LIN {X 0,Y 298.465,Z 418.303,A -85,B 0,C 180,E1 -16416.814,E2 -16416.814} C_VEL
LIN {X 0,Y 298.452,Z 418.307,A -85,B 0,C 180,E1 -16421.25,E2 -16421.25} C_VEL
LIN {X 0,Y 298.485,Z 418.303,A -85,B 0,C 180,E1 -16425.061,E2 -16425.061} C_VEL
LIN {X 0,Y 298.449,Z 418.307,A -85,B 0,C 180,E1 -16428.898,E2 -16428.898} C_VEL
LIN {X 0,Y 298.467,Z 418.307,A -85,B 0,C 180,E1 -16433.187,E2 -16433.187} C_VEL
LIN {X 0,Y 298.392,Z 418.317,A -85,B 0,C 180,E1 -16437.201,E2 -16437.201} C_VEL
LIN {X 0,Y 298.467,Z 418.305,A -85,B 0,C 180,E1 -16441.906,E2 -16441.906} C_VEL
LIN {X 0,Y 298.473,Z 418.306,A -85,B 0,C 180,E1 -16444.924,E2 -16444.924} C_VEL
LIN {X 0,Y 298.363,Z 418.483,A -85,B 0,C 180,E1 -16449.129,E2 -16449.129} C_VEL
LIN {X 0,Y 297.959,Z 422.878,A -85,B 0,C 180,E1 -16453.559,E2 -16453.559} C_VEL
LIN {X 0,Y 297.845,Z 425.727,A -85,B 0,C 180,E1 -16456.352,E2 -16456.352} C_VEL
LIN {X 0,Y 297.552,Z 430.816,A -85,B 0,C 180,E1 -16461.168,E2 -16461.168} C_VEL
LIN {X 0,Y 297.561,Z 431.032,A -85,B 0,C 180,E1 -16461.37,E2 -16461.37} C_VEL
LIN {X 0,Y 300.495,Z 443.519,A -85,B 0,C 180,E1 -16462.124,E2 -16462.124} C_VEL
LIN {X 0,Y 302.874,Z 456.628,A -85,B 0,C 180,E1 -16463.149,E2 -16463.149} C_VEL
LIN {X 0,Y 304.31,Z 467.202,A -85,B 0,C 180,E1 -16464.177,E2 -16464.177} C_VEL
LIN {X 0,Y 303.211,Z 477.949,A -85,B 0,C 180,E1 -16465.327,E2 -16465.327} C_VEL
LIN {X 0,Y 301.899,Z 489.013,A -85,B 0,C 180,E1 -16466.831,E2 -16466.831} C_VEL
LIN {X 0,Y 300.698,Z 497.91,A -85,B 0,C 180,E1 -16468.326,E2 -16468.326} C_VEL
LIN {X 0,Y 299.564,Z 506.081,A -85,B 0,C 180,E1 -16470,E2 -16470} C_VEL
LIN {X 0,Y 298.454,Z 514.101,A -85,B 0,C 180,E1 -16472.024,E2 -16472.024} C_VEL
LIN {X 0,Y 297.678,Z 520.511,A -85,B 0,C 180,E1 -16474.062,E2 -16474.062} C_VEL
LIN {X 0,Y 297.162,Z 525.845,A -85,B 0,C 180,E1 -16476.228,E2 -16476.228} C_VEL
LIN {X 0,Y 296.792,Z 529.552,A -85,B 0,C 180,E1 -16478.168,E2 -16478.168} C_VEL
LIN {X 0,Y 296.549,Z 531.596,A -85,B 0,C 180,E1 -16479.549,E2 -16479.549} C_VEL
LIN {X 0,Y 296.405,Z 533.217,A -85,B 0,C 180,E1 -16480.935,E2 -16480.935} C_VEL
LIN {X 0,Y 296.357,Z 535.085,A -85,B 0,C 180,E1 -16483.518,E2 -16483.518} C_VEL
LIN {X 0,Y 296.332,Z 535.507,A -85,B 0,C 180,E1 -16485.122,E2 -16485.122} C_VEL
LIN {X 0,Y 296.381,Z 535.459,A -85,B 0,C 180,E1 -16486.532,E2 -16486.532} C_VEL
LIN {X 0,Y 296.708,Z 534.552,A -85,B 0,C 180,E1 -16488.655,E2 -16488.655} C_VEL
LIN {X 0,Y 297.131,Z 532.679,A -85,B 0,C 180,E1 -16490.781,E2 -16490.781} C_VEL
LIN {X 0,Y 297.877,Z 529.561,A -85,B 0,C 180,E1 -16493.052,E2 -16493.052} C_VEL
LIN {X 0,Y 298.727,Z 525.744,A -85,B 0,C 180,E1 -16495.054,E2 -16495.054} C_VEL
LIN {X 0,Y 300.094,Z 519.861,A -85,B 0,C 180,E1 -16497.39,E2 -16497.39} C_VEL
LIN {X 0,Y 301.823,Z 512.406,A -85,B 0,C 180,E1 -16499.657,E2 -16499.657} C_VEL
LIN {X 0,Y 303.322,Z 505.485,A -85,B 0,C 180,E1 -16501.343,E2 -16501.343} C_VEL
LIN {X 0,Y 305.278,Z 496.379,A -85,B 0,C 180,E1 -16503.145,E2 -16503.145} C_VEL
LIN {X 0,Y 307.219,Z 486.66,A -85,B 0,C 180,E1 -16504.674,E2 -16504.674} C_VEL
LIN {X 0,Y 309.046,Z 475.83,A -85,B 0,C 180,E1 -16506.045,E2 -16506.045} C_VEL
LIN {X 0,Y 309.437,Z 473.03,A -85,B 0,C 180,E1 -16506.356,E2 -16506.356} C_VEL
LIN {X 0,Y 307.623,Z 462.047,A -85,B 0,C 180,E1 -16507.717,E2 -16507.717} C_VEL
LIN {X 0,Y 304.42,Z 449.779,A -85,B 0,C 180,E1 -16509.079,E2 -16509.079} C_VEL
LIN {X 0,Y 300.228,Z 437.616,A -85,B 0,C 180,E1 -16510.282,E2 -16510.282} C_VEL
LIN {X 0,Y 298.18,Z 432.147,A -85,B 0,C 180,E1 -16510.762,E2 -16510.762} C_VEL
LIN {X 0,Y 298.092,Z 431.637,A -85,B 0,C 180,E1 -16510.836,E2 -16510.836} C_VEL
LIN {X 0,Y 298.317,Z 429.506,A -85,B 0,C 180,E1 -16513.094,E2 -16513.094} C_VEL
LIN {X 0,Y 298.674,Z 426.006,A -85,B 0,C 180,E1 -16516.97,E2 -16516.97} C_VEL
LIN {X 0,Y 298.862,Z 424.41,A -85,B 0,C 180,E1 -16518.819,E2 -16518.819} C_VEL
LIN {X 0,Y 298.783,Z 421.553,A -85,B 0,C 180,E1 -16522.297,E2 -16522.297} C_VEL
LIN {X 0,Y 298.537,Z 419.047,A -85,B 0,C 180,E1 -16525.598,E2 -16525.598} C_VEL
LIN {X 0,Y 298.394,Z 418.32,A -85,B 0,C 180,E1 -16527.2,E2 -16527.2} C_VEL
LIN {X 0,Y 298.429,Z 418.312,A -85,B 0,C 180,E1 -16530.614,E2 -16530.614} C_VEL
LIN {X 0,Y 298.48,Z 418.307,A -85,B 0,C 180,E1 -16533.474,E2 -16533.474} C_VEL
LIN {X 0,Y 298.427,Z 418.313,A -85,B 0,C 180,E1 -16536.699,E2 -16536.699} C_VEL
LIN {X 0,Y 298.534,Z 418.296,A -85,B 0,C 180,E1 -16540.757,E2 -16540.757} C_VEL
LIN {X 0,Y 298.589,Z 418.291,A -85,B 0,C 180,E1 -16544.995,E2 -16544.995} C_VEL
LIN {X 0,Y 298.589,Z 418.287,A -85,B 0,C 180,E1 -16549.147,E2 -16549.147} C_VEL
LIN {X 0,Y 298.749,Z 418.27,A -85,B 0,C 180,E1 -16552.391,E2 -16552.391} C_VEL
LIN {X 0,Y 298.091,Z 418.355,A -85,B 0,C 180,E1 -16553.514,E2 -16553.514} C_VEL
LIN {X 0,Y 295.235,Z 418.71,A -85,B 0,C 180,E1 -16555.344,E2 -16555.344} C_VEL
LIN {X 0,Y 292.852,Z 419.006,A -85,B 0,C 180,E1 -16556.829,E2 -16556.829} C_VEL
LIN {X 0,Y 291.896,Z 419.127,A -85,B 0,C 180,E1 -16557.979,E2 -16557.979} C_VEL
LIN {X 0,Y 291.854,Z 419.128,A -85,B 0,C 180,E1 -16558.368,E2 -16558.368} C_VEL
LIN {X 0,Y 291.887,Z 419.128,A -85,B 0,C 180,E1 -16561.38,E2 -16561.38} C_VEL
LIN {X 0,Y 291.738,Z 419.14,A -85,B 0,C 180,E1 -16566.918,E2 -16566.918} C_VEL
LIN {X 0,Y 291.626,Z 419.161,A -85,B 0,C 180,E1 -16569.712,E2 -16569.712} C_VEL
LIN {X 0,Y 291.519,Z 419.172,A -85,B 0,C 180,E1 -16573.951,E2 -16573.951} C_VEL
LIN {X 0,Y 291.484,Z 419.179,A -85,B 0,C 180,E1 -16576.818,E2 -16576.818} C_VEL
LIN {X 0,Y 291.448,Z 419.185,A -85,B 0,C 180,E1 -16579.875,E2 -16579.875} C_VEL
LIN {X 0,Y 291.398,Z 419.19,A -85,B 0,C 180,E1 -16584.206,E2 -16584.206} C_VEL
LIN {X 0,Y 291.42,Z 419.187,A -85,B 0,C 180,E1 -16587.272,E2 -16587.272} C_VEL
LIN {X 0,Y 291.335,Z 419.197,A -85,B 0,C 180,E1 -16590.437,E2 -16590.437} C_VEL
LIN {X 0,Y 291.343,Z 419.194,A -85,B 0,C 180,E1 -16593.699,E2 -16593.699} C_VEL
LIN {X 0,Y 291.37,Z 419.185,A -85,B 0,C 180,E1 -16597.254,E2 -16597.254} C_VEL
LIN {X 0,Y 291.358,Z 419.241,A -85,B 0,C 180,E1 -16598.412,E2 -16598.412} C_VEL
LIN {X 0,Y 291.799,Z 422.011,A -85,B 0,C 180,E1 -16601.701,E2 -16601.701} C_VEL
LIN {X 0,Y 292.466,Z 425.825,A -85,B 0,C 180,E1 -16605.824,E2 -16605.824} C_VEL
LIN {X 0,Y 293.109,Z 429.691,A -85,B 0,C 180,E1 -16609.655,E2 -16609.655} C_VEL
LIN {X 0,Y 293.444,Z 433.625,A -85,B 0,C 180,E1 -16613.22,E2 -16613.22} C_VEL
LIN {X 0,Y 293.338,Z 435.615,A -85,B 0,C 180,E1 -16614.9,E2 -16614.9} C_VEL
LIN {X 0,Y 292.657,Z 439.593,A -85,B 0,C 180,E1 -16618.109,E2 -16618.109} C_VEL
LIN {X 0,Y 291.708,Z 445.236,A -85,B 0,C 180,E1 -16622.467,E2 -16622.467} C_VEL
LIN {X 0,Y 292.691,Z 448.629,A -85,B 0,C 180,E1 -16622.729,E2 -16622.729} C_VEL
LIN {X 0,Y 296.821,Z 462.357,A -85,B 0,C 180,E1 -16623.972,E2 -16623.972} C_VEL
LIN {X 0,Y 299.378,Z 474.172,A -85,B 0,C 180,E1 -16625.182,E2 -16625.182} C_VEL
LIN {X 0,Y 300.89,Z 486.394,A -85,B 0,C 180,E1 -16626.605,E2 -16626.605} C_VEL
LIN {X 0,Y 301.175,Z 494.957,A -85,B 0,C 180,E1 -16627.716,E2 -16627.716} C_VEL
LIN {X 0,Y 299.107,Z 505.649,A -85,B 0,C 180,E1 -16629.183,E2 -16629.183} C_VEL
LIN {X 0,Y 297.197,Z 514.413,A -85,B 0,C 180,E1 -16630.667,E2 -16630.667} C_VEL
LIN {X 0,Y 295.502,Z 522.486,A -85,B 0,C 180,E1 -16632.348,E2 -16632.348} C_VEL
LIN {X 0,Y 293.7,Z 530.437,A -85,B 0,C 180,E1 -16634.383,E2 -16634.383} C_VEL
LIN {X 0,Y 292.338,Z 535.848,A -85,B 0,C 180,E1 -16636.089,E2 -16636.089} C_VEL
LIN {X 0,Y 291.19,Z 541.166,A -85,B 0,C 180,E1 -16638.162,E2 -16638.162} C_VEL
LIN {X 0,Y 290.341,Z 545.336,A -85,B 0,C 180,E1 -16640.245,E2 -16640.245} C_VEL
LIN {X 0,Y 289.928,Z 547.557,A -85,B 0,C 180,E1 -16641.637,E2 -16641.637} C_VEL
LIN {X 0,Y 289.673,Z 549.306,A -85,B 0,C 180,E1 -16643.032,E2 -16643.032} C_VEL
LIN {X 0,Y 289.406,Z 551.603,A -85,B 0,C 180,E1 -16645.822,E2 -16645.822} C_VEL
LIN {X 0,Y 289.432,Z 552.172,A -85,B 0,C 180,E1 -16647.216,E2 -16647.216} C_VEL
LIN {X 0,Y 289.415,Z 552.31,A -85,B 0,C 180,E1 -16648.608,E2 -16648.608} C_VEL
LIN {X 0,Y 289.438,Z 552.054,A -85,B 0,C 180,E1 -16650,E2 -16650} C_VEL
LIN {X 0,Y 289.421,Z 551.408,A -85,B 0,C 180,E1 -16651.391,E2 -16651.391} C_VEL
LIN {X 0,Y 289.467,Z 550.372,A -85,B 0,C 180,E1 -16652.783,E2 -16652.783} C_VEL
LIN {X 0,Y 289.434,Z 548.879,A -85,B 0,C 180,E1 -16654.177,E2 -16654.177} C_VEL
LIN {X 0,Y 289.554,Z 545.838,A -85,B 0,C 180,E1 -16656.27,E2 -16656.27} C_VEL
LIN {X 0,Y 289.851,Z 541.724,A -85,B 0,C 180,E1 -16658.365,E2 -16658.365} C_VEL
LIN {X 0,Y 290.47,Z 535.4,A -85,B 0,C 180,E1 -16660.807,E2 -16660.807} C_VEL
LIN {X 0,Y 291.304,Z 528.501,A -85,B 0,C 180,E1 -16662.894,E2 -16662.894} C_VEL
LIN {X 0,Y 292.264,Z 521.451,A -85,B 0,C 180,E1 -16664.624,E2 -16664.624} C_VEL
LIN {X 0,Y 293.456,Z 512.95,A -85,B 0,C 180,E1 -16666.343,E2 -16666.343} C_VEL
LIN {X 0,Y 294.727,Z 502.406,A -85,B 0,C 180,E1 -16668.058,E2 -16668.058} C_VEL
LIN {X 0,Y 296.106,Z 491.99,A -85,B 0,C 180,E1 -16669.407,E2 -16669.407} C_VEL
LIN {X 0,Y 296.167,Z 487.329,A -85,B 0,C 180,E1 -16669.944,E2 -16669.944} C_VEL
LIN {X 0,Y 295.093,Z 475.372,A -85,B 0,C 180,E1 -16671.174,E2 -16671.174} C_VEL
LIN {X 0,Y 293.48,Z 462.982,A -85,B 0,C 180,E1 -16672.178,E2 -16672.178} C_VEL
LIN {X 0,Y 291.441,Z 450.758,A -85,B 0,C 180,E1 -16672.935,E2 -16672.935} C_VEL
LIN {X 0,Y 290.549,Z 445.893,A -85,B 0,C 180,E1 -16673.194,E2 -16673.194} C_VEL
LIN {X 0,Y 291.111,Z 440.04,A -85,B 0,C 180,E1 -16677.302,E2 -16677.302} C_VEL
LIN {X 0,Y 292.02,Z 433.549,A -85,B 0,C 180,E1 -16681.969,E2 -16681.969} C_VEL
LIN {X 0,Y 292.587,Z 429.133,A -85,B 0,C 180,E1 -16685.245,E2 -16685.245} C_VEL
LIN {X 0,Y 292.659,Z 426.105,A -85,B 0,C 180,E1 -16687.583,E2 -16687.583} C_VEL
LIN {X 0,Y 291.783,Z 421.133,A -85,B 0,C 180,E1 -16691.696,E2 -16691.696} C_VEL
LIN {X 0,Y 291.441,Z 419.183,A -85,B 0,C 180,E1 -16693.518,E2 -16693.518} C_VEL
LIN {X 0,Y 291.337,Z 419.196,A -85,B 0,C 180,E1 -16697.51,E2 -16697.51} C_VEL
LIN {X 0,Y 291.349,Z 419.196,A -85,B 0,C 180,E1 -16701.157,E2 -16701.157} C_VEL
LIN {X 0,Y 291.357,Z 419.193,A -85,B 0,C 180,E1 -16704.625,E2 -16704.625} C_VEL
LIN {X 0,Y 291.367,Z 419.188,A -85,B 0,C 180,E1 -16707.95,E2 -16707.95} C_VEL
LIN {X 0,Y 291.377,Z 419.184,A -85,B 0,C 180,E1 -16711.158,E2 -16711.158} C_VEL
LIN {X 0,Y 291.411,Z 419.181,A -85,B 0,C 180,E1 -16714.271,E2 -16714.271} C_VEL
LIN {X 0,Y 291.376,Z 419.188,A -85,B 0,C 180,E1 -16717.299,E2 -16717.299} C_VEL
LIN {X 0,Y 291.452,Z 419.178,A -85,B 0,C 180,E1 -16720.269,E2 -16720.269} C_VEL
LIN {X 0,Y 291.51,Z 419.167,A -85,B 0,C 180,E1 -16724.652,E2 -16724.652} C_VEL
LIN {X 0,Y 291.53,Z 419.17,A -85,B 0,C 180,E1 -16728.88,E2 -16728.88} C_VEL
LIN {X 0,Y 291.704,Z 419.146,A -85,B 0,C 180,E1 -16731.688,E2 -16731.688} C_VEL
LIN {X 0,Y 291.627,Z 419.154,A -85,B 0,C 180,E1 -16734.468,E2 -16734.468} C_VEL
LIN {X 0,Y 291.884,Z 419.122,A -85,B 0,C 180,E1 -16738.62,E2 -16738.62} C_VEL
LIN {X 0,Y 291.884,Z 419.122,A -85,B 0,C 180,E1 -16741.379,E2 -16741.379} C_VEL
LIN {X 0,Y 291.739,Z 419.14,A -85,B 0,C 180,E1 -16746.918,E2 -16746.918} C_VEL
LIN {X 0,Y 291.623,Z 419.152,A -85,B 0,C 180,E1 -16749.712,E2 -16749.712} C_VEL
LIN {X 0,Y 291.515,Z 419.168,A -85,B 0,C 180,E1 -16753.95,E2 -16753.95} C_VEL
LIN {X 0,Y 291.48,Z 419.174,A -85,B 0,C 180,E1 -16756.818,E2 -16756.818} C_VEL
LIN {X 0,Y 291.444,Z 419.183,A -85,B 0,C 180,E1 -16759.875,E2 -16759.875} C_VEL
LIN {X 0,Y 291.394,Z 419.188,A -85,B 0,C 180,E1 -16764.206,E2 -16764.206} C_VEL
LIN {X 0,Y 291.417,Z 419.183,A -85,B 0,C 180,E1 -16767.272,E2 -16767.272} C_VEL
LIN {X 0,Y 291.333,Z 419.193,A -85,B 0,C 180,E1 -16770.437,E2 -16770.437} C_VEL
LIN {X 0,Y 291.34,Z 419.196,A -85,B 0,C 180,E1 -16773.699,E2 -16773.699} C_VEL
LIN {X 0,Y 291.4,Z 419.185,A -85,B 0,C 180,E1 -16777.262,E2 -16777.262} C_VEL
LIN {X 0,Y 291.402,Z 419.184,A -85,B 0,C 180,E1 -16780.631,E2 -16780.631} C_VEL
LIN {X 0,Y 291.402,Z 419.184,A -85,B 0,C 180,E1 -16784.38,E2 -16784.38} C_VEL
LIN {X 0,Y 291.385,Z 419.186,A -85,B 0,C 180,E1 -16788.391,E2 -16788.391} C_VEL
LIN {X 0,Y 291.382,Z 419.189,A -85,B 0,C 180,E1 -16791.164,E2 -16791.164} C_VEL
LIN {X 0,Y 291.383,Z 419.186,A -85,B 0,C 180,E1 -16794.63,E2 -16794.63} C_VEL
LIN {X 0,Y 291.369,Z 419.189,A -85,B 0,C 180,E1 -16797.951,E2 -16797.951} C_VEL
LIN {X 0,Y 291.383,Z 419.191,A -85,B 0,C 180,E1 -16801.159,E2 -16801.159} C_VEL
LIN {X 0,Y 291.412,Z 419.183,A -85,B 0,C 180,E1 -16804.272,E2 -16804.272} C_VEL
LIN {X 0,Y 291.333,Z 419.198,A -85,B 0,C 180,E1 -16807.296,E2 -16807.296} C_VEL
LIN {X 0,Y 291.326,Z 419.259,A -85,B 0,C 180,E1 -16808.971,E2 -16808.971} C_VEL
LIN {X 0,Y 290.92,Z 423.325,A -85,B 0,C 180,E1 -16813.149,E2 -16813.149} C_VEL
LIN {X 0,Y 290.813,Z 426.158,A -85,B 0,C 180,E1 -16816.016,E2 -16816.016} C_VEL
LIN {X 0,Y 290.487,Z 431.194,A -85,B 0,C 180,E1 -16820.909,E2 -16820.909} C_VEL
LIN {X 0,Y 293.642,Z 444.431,A -85,B 0,C 180,E1 -16821.744,E2 -16821.744} C_VEL
LIN {X 0,Y 295.894,Z 456.669,A -85,B 0,C 180,E1 -16822.732,E2 -16822.732} C_VEL
LIN {X 0,Y 297.439,Z 468.377,A -85,B 0,C 180,E1 -16823.903,E2 -16823.903} C_VEL
LIN {X 0,Y 296.107,Z 480.124,A -85,B 0,C 180,E1 -16825.235,E2 -16825.235} C_VEL
LIN {X 0,Y 294.762,Z 490.697,A -85,B 0,C 180,E1 -16826.754,E2 -16826.754} C_VEL
LIN {X 0,Y 293.573,Z 499.343,A -85,B 0,C 180,E1 -16828.286,E2 -16828.286} C_VEL
LIN {X 0,Y 292.435,Z 507.31,A -85,B 0,C 180,E1 -16830,E2 -16830} C_VEL
LIN {X 0,Y 291.307,Z 515.11,A -85,B 0,C 180,E1 -16832.074,E2 -16832.074} C_VEL
LIN {X 0,Y 290.54,Z 521.342,A -85,B 0,C 180,E1 -16834.162,E2 -16834.162} C_VEL
LIN {X 0,Y 290.026,Z 526.838,A -85,B 0,C 180,E1 -16836.525,E2 -16836.525} C_VEL
LIN {X 0,Y 289.668,Z 530.129,A -85,B 0,C 180,E1 -16838.371,E2 -16838.371} C_VEL
LIN {X 0,Y 289.437,Z 532.113,A -85,B 0,C 180,E1 -16839.786,E2 -16839.786} C_VEL
LIN {X 0,Y 289.309,Z 533.671,A -85,B 0,C 180,E1 -16841.206,E2 -16841.206} C_VEL
LIN {X 0,Y 289.267,Z 535.298,A -85,B 0,C 180,E1 -16843.631,E2 -16843.631} C_VEL
LIN {X 0,Y 289.249,Z 535.745,A -85,B 0,C 180,E1 -16845.502,E2 -16845.502} C_VEL
LIN {X 0,Y 289.343,Z 535.61,A -85,B 0,C 180,E1 -16846.946,E2 -16846.946} C_VEL
LIN {X 0,Y 289.654,Z 534.762,A -85,B 0,C 180,E1 -16848.867,E2 -16848.867} C_VEL
LIN {X 0,Y 290.176,Z 532.62,A -85,B 0,C 180,E1 -16851.303,E2 -16851.303} C_VEL
LIN {X 0,Y 290.911,Z 529.789,A -85,B 0,C 180,E1 -16853.361,E2 -16853.361} C_VEL
LIN {X 0,Y 291.95,Z 525.412,A -85,B 0,C 180,E1 -16855.677,E2 -16855.677} C_VEL
LIN {X 0,Y 293.562,Z 518.888,A -85,B 0,C 180,E1 -16858.223,E2 -16858.223} C_VEL
LIN {X 0,Y 295.311,Z 511.768,A -85,B 0,C 180,E1 -16860.369,E2 -16860.369} C_VEL
LIN {X 0,Y 297.053,Z 504.313,A -85,B 0,C 180,E1 -16862.163,E2 -16862.163} C_VEL
LIN {X 0,Y 299.057,Z 495.217,A -85,B 0,C 180,E1 -16863.927,E2 -16863.927} C_VEL
LIN {X 0,Y 301.046,Z 485.307,A -85,B 0,C 180,E1 -16865.474,E2 -16865.474} C_VEL
LIN {X 0,Y 302.799,Z 475.524,A -85,B 0,C 180,E1 -16866.702,E2 -16866.702} C_VEL
LIN {X 0,Y 302.479,Z 471.193,A -85,B 0,C 180,E1 -16867.27,E2 -16867.27} C_VEL
LIN {X 0,Y 300.73,Z 461.738,A -85,B 0,C 180,E1 -16868.474,E2 -16868.474} C_VEL
LIN {X 0,Y 297.539,Z 449.751,A -85,B 0,C 180,E1 -16869.855,E2 -16869.855} C_VEL
LIN {X 0,Y 293.304,Z 437.857,A -85,B 0,C 180,E1 -16871.096,E2 -16871.096} C_VEL
LIN {X 0,Y 291.268,Z 432.706,A -85,B 0,C 180,E1 -16871.583,E2 -16871.583} C_VEL
LIN {X 0,Y 291.127,Z 431.864,A -85,B 0,C 180,E1 -16871.669,E2 -16871.669} C_VEL
LIN {X 0,Y 291.51,Z 428.287,A -85,B 0,C 180,E1 -16875.641,E2 -16875.641} C_VEL
LIN {X 0,Y 291.85,Z 425.048,A -85,B 0,C 180,E1 -16879.445,E2 -16879.445} C_VEL
LIN {X 0,Y 291.775,Z 422.264,A -85,B 0,C 180,E1 -16882.974,E2 -16882.974} C_VEL
LIN {X 0,Y 291.431,Z 419.831,A -85,B 0,C 180,E1 -16886.313,E2 -16886.313} C_VEL
LIN {X 0,Y 291.371,Z 419.194,A -85,B 0,C 180,E1 -16887.951,E2 -16887.951} C_VEL
LIN {X 0,Y 291.379,Z 419.19,A -85,B 0,C 180,E1 -16891.158,E2 -16891.158} C_VEL
LIN {X 0,Y 291.412,Z 419.186,A -85,B 0,C 180,E1 -16894.272,E2 -16894.272} C_VEL
LIN {X 0,Y 291.37,Z 419.191,A -85,B 0,C 180,E1 -16897.299,E2 -16897.299} C_VEL
LIN {X 0,Y 291.454,Z 419.178,A -85,B 0,C 180,E1 -16900.27,E2 -16900.27} C_VEL
LIN {X 0,Y 291.536,Z 419.172,A -85,B 0,C 180,E1 -16904.634,E2 -16904.634} C_VEL
LIN {X 0,Y 291.532,Z 419.166,A -85,B 0,C 180,E1 -16908.881,E2 -16908.881} C_VEL
LIN {X 0,Y 291.702,Z 419.147,A -85,B 0,C 180,E1 -16912.398,E2 -16912.398} C_VEL
LIN {X 0,Y 291.785,Z 419.138,A -85,B 0,C 180,E1 -16917.239,E2 -16917.239} C_VEL
LIN {X 0,Y 291.854,Z 419.128,A -85,B 0,C 180,E1 -16918.368,E2 -16918.368} C_VEL
LIN {X 0,Y 291.242,Z 419.21,A -85,B 0,C 180,E1 -16919.521,E2 -16919.521} C_VEL
LIN {X 0,Y 288.261,Z 419.585,A -85,B 0,C 180,E1 -16921.391,E2 -16921.391} C_VEL
LIN {X 0,Y 285.684,Z 419.903,A -85,B 0,C 180,E1 -16922.911,E2 -16922.911} C_VEL
LIN {X 0,Y 284.588,Z 420.036,A -85,B 0,C 180,E1 -16924.093,E2 -16924.093} C_VEL
LIN {X 0,Y 284.509,Z 420.044,A -85,B 0,C 180,E1 -16924.495,E2 -16924.495} C_VEL
LIN {X 0,Y 284.69,Z 420.017,A -85,B 0,C 180,E1 -16927.09,E2 -16927.09} C_VEL
LIN {X 0,Y 284.563,Z 420.039,A -85,B 0,C 180,E1 -16929.956,E2 -16929.956} C_VEL
LIN {X 0,Y 284.479,Z 420.05,A -85,B 0,C 180,E1 -16934.303,E2 -16934.303} C_VEL
LIN {X 0,Y 284.422,Z 420.058,A -85,B 0,C 180,E1 -16937.249,E2 -16937.249} C_VEL
LIN {X 0,Y 284.376,Z 420.066,A -85,B 0,C 180,E1 -16940.243,E2 -16940.243} C_VEL
LIN {X 0,Y 284.366,Z 420.066,A -85,B 0,C 180,E1 -16943.876,E2 -16943.876} C_VEL
LIN {X 0,Y 284.395,Z 420.062,A -85,B 0,C 180,E1 -16947.174,E2 -16947.174} C_VEL
LIN {X 0,Y 284.294,Z 420.073,A -85,B 0,C 180,E1 -16951.275,E2 -16951.275} C_VEL
LIN {X 0,Y 284.339,Z 420.064,A -85,B 0,C 180,E1 -16955.349,E2 -16955.349} C_VEL
LIN {X 0,Y 284.355,Z 420.241,A -85,B 0,C 180,E1 -16957.731,E2 -16957.731} C_VEL
LIN {X 0,Y 284.687,Z 422.109,A -85,B 0,C 180,E1 -16960.068,E2 -16960.068} C_VEL
LIN {X 0,Y 285.292,Z 425.882,A -85,B 0,C 180,E1 -16964.407,E2 -16964.407} C_VEL
LIN {X 0,Y 285.931,Z 429.723,A -85,B 0,C 180,E1 -16968.422,E2 -16968.422} C_VEL
LIN {X 0,Y 286.429,Z 433.64,A -85,B 0,C 180,E1 -16972.164,E2 -16972.164} C_VEL
LIN {X 0,Y 286.395,Z 435.785,A -85,B 0,C 180,E1 -16974.077,E2 -16974.077} C_VEL
LIN {X 0,Y 285.824,Z 439.581,A -85,B 0,C 180,E1 -16977.252,E2 -16977.252} C_VEL
LIN {X 0,Y 284.843,Z 445.097,A -85,B 0,C 180,E1 -16981.6,E2 -16981.6} C_VEL
LIN {X 0,Y 285.725,Z 448.198,A -85,B 0,C 180,E1 -16981.843,E2 -16981.843} C_VEL
LIN {X 0,Y 289.583,Z 460.533,A -85,B 0,C 180,E1 -16983.01,E2 -16983.01} C_VEL
LIN {X 0,Y 292.28,Z 471.987,A -85,B 0,C 180,E1 -16984.22,E2 -16984.22} C_VEL
LIN {X 0,Y 293.892,Z 482.991,A -85,B 0,C 180,E1 -16985.509,E2 -16985.509} C_VEL
LIN {X 0,Y 294.589,Z 492.921,A -85,B 0,C 180,E1 -16986.819,E2 -16986.819} C_VEL
LIN {X 0,Y 294.298,Z 498.108,A -85,B 0,C 180,E1 -16987.537,E2 -16987.537} C_VEL
LIN {X 0,Y 292.009,Z 508.219,A -85,B 0,C 180,E1 -16989.022,E2 -16989.022} C_VEL
LIN {X 0,Y 289.773,Z 518.139,A -85,B 0,C 180,E1 -16990.889,E2 -16990.889} C_VEL
LIN {X 0,Y 287.769,Z 526.893,A -85,B 0,C 180,E1 -16992.958,E2 -16992.958} C_VEL
LIN {X 0,Y 286.016,Z 533.945,A -85,B 0,C 180,E1 -16995.048,E2 -16995.048} C_VEL
LIN {X 0,Y 284.539,Z 539.599,A -85,B 0,C 180,E1 -16997.156,E2 -16997.156} C_VEL
LIN {X 0,Y 283.566,Z 544.076,A -85,B 0,C 180,E1 -16999.287,E2 -16999.287} C_VEL
LIN {X 0,Y 282.896,Z 547.498,A -85,B 0,C 180,E1 -17001.428,E2 -17001.428} C_VEL
LIN {X 0,Y 282.409,Z 550.527,A -85,B 0,C 180,E1 -17004.287,E2 -17004.287} C_VEL
LIN {X 0,Y 282.316,Z 551.457,A -85,B 0,C 180,E1 -17005.717,E2 -17005.717} C_VEL
LIN {X 0,Y 282.338,Z 551.989,A -85,B 0,C 180,E1 -17007.146,E2 -17007.146} C_VEL
LIN {X 0,Y 282.337,Z 552.094,A -85,B 0,C 180,E1 -17008.573,E2 -17008.573} C_VEL
LIN {X 0,Y 282.358,Z 551.814,A -85,B 0,C 180,E1 -17010,E2 -17010} C_VEL
LIN {X 0,Y 282.344,Z 551.145,A -85,B 0,C 180,E1 -17011.426,E2 -17011.426} C_VEL
LIN {X 0,Y 282.372,Z 550.074,A -85,B 0,C 180,E1 -17012.853,E2 -17012.853} C_VEL
LIN {X 0,Y 282.403,Z 546.964,A -85,B 0,C 180,E1 -17015.461,E2 -17015.461} C_VEL
LIN {X 0,Y 282.673,Z 542.784,A -85,B 0,C 180,E1 -17017.859,E2 -17017.859} C_VEL
LIN {X 0,Y 283.136,Z 537.838,A -85,B 0,C 180,E1 -17020.006,E2 -17020.006} C_VEL
LIN {X 0,Y 283.818,Z 531.595,A -85,B 0,C 180,E1 -17022.15,E2 -17022.15} C_VEL
LIN {X 0,Y 284.984,Z 523.807,A -85,B 0,C 180,E1 -17024.276,E2 -17024.276} C_VEL
LIN {X 0,Y 286.319,Z 514.309,A -85,B 0,C 180,E1 -17026.335,E2 -17026.335} C_VEL
LIN {X 0,Y 287.606,Z 504.078,A -85,B 0,C 180,E1 -17028.116,E2 -17028.116} C_VEL
LIN {X 0,Y 288.975,Z 493.777,A -85,B 0,C 180,E1 -17029.536,E2 -17029.536} C_VEL
LIN {X 0,Y 289.334,Z 489.38,A -85,B 0,C 180,E1 -17030.065,E2 -17030.065} C_VEL
LIN {X 0,Y 288.333,Z 477.389,A -85,B 0,C 180,E1 -17031.374,E2 -17031.374} C_VEL
LIN {X 0,Y 286.715,Z 464.217,A -85,B 0,C 180,E1 -17032.518,E2 -17032.518} C_VEL
LIN {X 0,Y 284.708,Z 452.031,A -85,B 0,C 180,E1 -17033.327,E2 -17033.327} C_VEL
LIN {X 0,Y 283.549,Z 445.675,A -85,B 0,C 180,E1 -17033.682,E2 -17033.682} C_VEL
LIN {X 0,Y 284.13,Z 439.676,A -85,B 0,C 180,E1 -17038.031,E2 -17038.031} C_VEL
LIN {X 0,Y 284.978,Z 434.259,A -85,B 0,C 180,E1 -17042.02,E2 -17042.02} C_VEL
LIN {X 0,Y 285.578,Z 429.454,A -85,B 0,C 180,E1 -17045.696,E2 -17045.696} C_VEL
LIN {X 0,Y 285.548,Z 426.525,A -85,B 0,C 180,E1 -17048.038,E2 -17048.038} C_VEL
LIN {X 0,Y 284.684,Z 421.629,A -85,B 0,C 180,E1 -17052.216,E2 -17052.216} C_VEL
LIN {X 0,Y 284.363,Z 420.064,A -85,B 0,C 180,E1 -17053.788,E2 -17053.788} C_VEL
LIN {X 0,Y 284.279,Z 420.073,A -85,B 0,C 180,E1 -17058.125,E2 -17058.125} C_VEL
LIN {X 0,Y 284.319,Z 420.068,A -85,B 0,C 180,E1 -17062.277,E2 -17062.277} C_VEL
LIN {X 0,Y 284.304,Z 420.07,A -85,B 0,C 180,E1 -17065.35,E2 -17065.35} C_VEL
LIN {X 0,Y 284.291,Z 420.074,A -85,B 0,C 180,E1 -17068.725,E2 -17068.725} C_VEL
LIN {X 0,Y 284.393,Z 420.055,A -85,B 0,C 180,E1 -17072.826,E2 -17072.826} C_VEL
LIN {X 0,Y 284.361,Z 420.065,A -85,B 0,C 180,E1 -17076.706,E2 -17076.706} C_VEL
LIN {X 0,Y 284.396,Z 420.052,A -85,B 0,C 180,E1 -17081.261,E2 -17081.261} C_VEL
LIN {X 0,Y 284.463,Z 420.044,A -85,B 0,C 180,E1 -17085.696,E2 -17085.696} C_VEL
LIN {X 0,Y 284.56,Z 420.038,A -85,B 0,C 180,E1 -17090.044,E2 -17090.044} C_VEL
LIN {X 0,Y 284.694,Z 420.018,A -85,B 0,C 180,E1 -17092.91,E2 -17092.91} C_VEL
LIN {X 0,Y 284.85,Z 419.997,A -85,B 0,C 180,E1 -17098.586,E2 -17098.586} C_VEL
LIN {X 0,Y 284.85,Z 419.999,A -85,B 0,C 180,E1 -17101.414,E2 -17101.414} C_VEL
LIN {X 0,Y 284.692,Z 420.018,A -85,B 0,C 180,E1 -17107.09,E2 -17107.09} C_VEL
LIN {X 0,Y 284.56,Z 420.032,A -85,B 0,C 180,E1 -17109.955,E2 -17109.955} C_VEL
LIN {X 0,Y 284.471,Z 420.048,A -85,B 0,C 180,E1 -17114.303,E2 -17114.303} C_VEL
LIN {X 0,Y 284.419,Z 420.054,A -85,B 0,C 180,E1 -17117.249,E2 -17117.249} C_VEL
LIN {X 0,Y 284.372,Z 420.061,A -85,B 0,C 180,E1 -17120.242,E2 -17120.242} C_VEL
LIN {X 0,Y 284.363,Z 420.064,A -85,B 0,C 180,E1 -17123.876,E2 -17123.876} C_VEL
LIN {X 0,Y 284.391,Z 420.057,A -85,B 0,C 180,E1 -17127.174,E2 -17127.174} C_VEL
LIN {X 0,Y 284.293,Z 420.07,A -85,B 0,C 180,E1 -17131.274,E2 -17131.274} C_VEL
LIN {X 0,Y 284.357,Z 420.062,A -85,B 0,C 180,E1 -17135.355,E2 -17135.355} C_VEL
LIN {X 0,Y 284.333,Z 420.066,A -85,B 0,C 180,E1 -17138.165,E2 -17138.165} C_VEL
LIN {X 0,Y 284.34,Z 420.065,A -85,B 0,C 180,E1 -17142.142,E2 -17142.142} C_VEL
LIN {X 0,Y 284.349,Z 420.063,A -85,B 0,C 180,E1 -17146.209,E2 -17146.209} C_VEL
LIN {X 0,Y 284.348,Z 420.064,A -85,B 0,C 180,E1 -17150.014,E2 -17150.014} C_VEL
LIN {X 0,Y 284.352,Z 420.065,A -85,B 0,C 180,E1 -17153.618,E2 -17153.618} C_VEL
LIN {X 0,Y 284.305,Z 420.072,A -85,B 0,C 180,E1 -17157.19,E2 -17157.19} C_VEL
LIN {X 0,Y 284.357,Z 420.062,A -85,B 0,C 180,E1 -17160.377,E2 -17160.377} C_VEL
LIN {X 0,Y 284.376,Z 420.062,A -85,B 0,C 180,E1 -17163.587,E2 -17163.587} C_VEL
LIN {X 0,Y 284.307,Z 420.071,A -85,B 0,C 180,E1 -17166.703,E2 -17166.703} C_VEL
LIN {X 0,Y 284.29,Z 420.209,A -85,B 0,C 180,E1 -17168.995,E2 -17168.995} C_VEL
LIN {X 0,Y 283.897,Z 423.761,A -85,B 0,C 180,E1 -17172.719,E2 -17172.719} C_VEL
LIN {X 0,Y 283.774,Z 426.632,A -85,B 0,C 180,E1 -17175.661,E2 -17175.661} C_VEL
LIN {X 0,Y 283.457,Z 431.518,A -85,B 0,C 180,E1 -17180.44,E2 -17180.44} C_VEL
LIN {X 0,Y 286.668,Z 444.43,A -85,B 0,C 180,E1 -17181.282,E2 -17181.282} C_VEL
LIN {X 0,Y 288.979,Z 457.242,A -85,B 0,C 180,E1 -17182.346,E2 -17182.346} C_VEL
LIN {X 0,Y 290.552,Z 469.113,A -85,B 0,C 180,E1 -17183.577,E2 -17183.577} C_VEL
LIN {X 0,Y 289.187,Z 480.782,A -85,B 0,C 180,E1 -17184.946,E2 -17184.946} C_VEL
LIN {X 0,Y 287.802,Z 491.281,A -85,B 0,C 180,E1 -17186.5,E2 -17186.5} C_VEL
LIN {X 0,Y 286.455,Z 500.744,A -85,B 0,C 180,E1 -17188.243,E2 -17188.243} C_VEL
LIN {X 0,Y 285.11,Z 509.852,A -85,B 0,C 180,E1 -17190.353,E2 -17190.353} C_VEL
LIN {X 0,Y 284.079,Z 517.193,A -85,B 0,C 180,E1 -17192.482,E2 -17192.482} C_VEL
LIN {X 0,Y 283.411,Z 522.168,A -85,B 0,C 180,E1 -17194.267,E2 -17194.267} C_VEL
LIN {X 0,Y 282.94,Z 527.16,A -85,B 0,C 180,E1 -17196.503,E2 -17196.503} C_VEL
LIN {X 0,Y 282.535,Z 530.705,A -85,B 0,C 180,E1 -17198.583,E2 -17198.583} C_VEL
LIN {X 0,Y 282.321,Z 532.63,A -85,B 0,C 180,E1 -17200.035,E2 -17200.035} C_VEL
LIN {X 0,Y 282.194,Z 534.081,A -85,B 0,C 180,E1 -17201.492,E2 -17201.492} C_VEL
LIN {X 0,Y 282.162,Z 535.506,A -85,B 0,C 180,E1 -17203.737,E2 -17203.737} C_VEL
LIN {X 0,Y 282.163,Z 535.967,A -85,B 0,C 180,E1 -17205.901,E2 -17205.901} C_VEL
LIN {X 0,Y 282.304,Z 535.734,A -85,B 0,C 180,E1 -17207.382,E2 -17207.382} C_VEL
LIN {X 0,Y 282.609,Z 534.972,A -85,B 0,C 180,E1 -17209.093,E2 -17209.093} C_VEL
LIN {X 0,Y 283.24,Z 532.52,A -85,B 0,C 180,E1 -17211.851,E2 -17211.851} C_VEL
LIN {X 0,Y 283.938,Z 530.039,A -85,B 0,C 180,E1 -17213.678,E2 -17213.678} C_VEL
LIN {X 0,Y 284.802,Z 526.624,A -85,B 0,C 180,E1 -17215.584,E2 -17215.584} C_VEL
LIN {X 0,Y 286.202,Z 521.346,A -85,B 0,C 180,E1 -17217.87,E2 -17217.87} C_VEL
LIN {X 0,Y 287.883,Z 514.925,A -85,B 0,C 180,E1 -17220.03,E2 -17220.03} C_VEL
LIN {X 0,Y 289.94,Z 506.595,A -85,B 0,C 180,E1 -17222.226,E2 -17222.226} C_VEL
LIN {X 0,Y 291.963,Z 498.017,A -85,B 0,C 180,E1 -17224.032,E2 -17224.032} C_VEL
LIN {X 0,Y 294.179,Z 488.217,A -85,B 0,C 180,E1 -17225.682,E2 -17225.682} C_VEL
LIN {X 0,Y 296.245,Z 477.059,A -85,B 0,C 180,E1 -17227.174,E2 -17227.174} C_VEL
LIN {X 0,Y 296.07,Z 473.359,A -85,B 0,C 180,E1 -17227.683,E2 -17227.683} C_VEL
LIN {X 0,Y 294.624,Z 464.735,A -85,B 0,C 180,E1 -17228.854,E2 -17228.854} C_VEL
LIN {X 0,Y 291.566,Z 452.701,A -85,B 0,C 180,E1 -17230.334,E2 -17230.334} C_VEL
LIN {X 0,Y 287.768,Z 441.556,A -85,B 0,C 180,E1 -17231.582,E2 -17231.582} C_VEL
LIN {X 0,Y 284.317,Z 432.883,A -85,B 0,C 180,E1 -17232.476,E2 -17232.476} C_VEL
LIN {X 0,Y 284.178,Z 432.102,A -85,B 0,C 180,E1 -17232.559,E2 -17232.559} C_VEL
LIN {X 0,Y 284.571,Z 428.873,A -85,B 0,C 180,E1 -17236.25,E2 -17236.25} C_VEL
LIN {X 0,Y 284.843,Z 425.872,A -85,B 0,C 180,E1 -17239.895,E2 -17239.895} C_VEL
LIN {X 0,Y 284.691,Z 423.007,A -85,B 0,C 180,E1 -17243.668,E2 -17243.668} C_VEL
LIN {X 0,Y 284.35,Z 420.555,A -85,B 0,C 180,E1 -17247.175,E2 -17247.175} C_VEL
LIN {X 0,Y 284.294,Z 420.076,A -85,B 0,C 180,E1 -17248.726,E2 -17248.726} C_VEL
LIN {X 0,Y 284.394,Z 420.061,A -85,B 0,C 180,E1 -17252.826,E2 -17252.826} C_VEL
LIN {X 0,Y 284.329,Z 420.069,A -85,B 0,C 180,E1 -17256.704,E2 -17256.704} C_VEL
LIN {X 0,Y 284.399,Z 420.059,A -85,B 0,C 180,E1 -17261.262,E2 -17261.262} C_VEL
LIN {X 0,Y 284.474,Z 420.052,A -85,B 0,C 180,E1 -17264.47,E2 -17264.47} C_VEL
LIN {X 0,Y 284.484,Z 420.045,A -85,B 0,C 180,E1 -17268.602,E2 -17268.602} C_VEL
LIN {X 0,Y 284.655,Z 420.027,A -85,B 0,C 180,E1 -17271.481,E2 -17271.481} C_VEL
LIN {X 0,Y 284.597,Z 420.035,A -85,B 0,C 180,E1 -17274.331,E2 -17274.331} C_VEL
LIN {X 0,Y 284.851,Z 420.002,A -85,B 0,C 180,E1 -17278.586,E2 -17278.586} C_VEL
LIN {X 0,Y 284.853,Z 420.004,A -85,B 0,C 180,E1 -17281.414,E2 -17281.414} C_VEL
LIN {X 0,Y 284.509,Z 420.044,A -85,B 0,C 180,E1 -17284.495,E2 -17284.495} C_VEL
LIN {X 0,Y 283.876,Z 420.126,A -85,B 0,C 180,E1 -17285.678,E2 -17285.678} C_VEL
LIN {X 0,Y 281.061,Z 420.473,A -85,B 0,C 180,E1 -17287.606,E2 -17287.606} C_VEL
LIN {X 0,Y 278.632,Z 420.778,A -85,B 0,C 180,E1 -17289.171,E2 -17289.171} C_VEL
LIN {X 0,Y 277.558,Z 420.911,A -85,B 0,C 180,E1 -17290.384,E2 -17290.384} C_VEL
LIN {X 0,Y 277.454,Z 420.922,A -85,B 0,C 180,E1 -17290.795,E2 -17290.795} C_VEL
LIN {X 0,Y 277.432,Z 420.93,A -85,B 0,C 180,E1 -17294.675,E2 -17294.675} C_VEL
LIN {X 0,Y 277.342,Z 420.941,A -85,B 0,C 180,E1 -17299.234,E2 -17299.234} C_VEL
LIN {X 0,Y 277.317,Z 420.944,A -85,B 0,C 180,E1 -17304.171,E2 -17304.171} C_VEL
LIN {X 0,Y 277.324,Z 420.943,A -85,B 0,C 180,E1 -17307.506,E2 -17307.506} C_VEL
LIN {X 0,Y 277.27,Z 420.949,A -85,B 0,C 180,E1 -17310.482,E2 -17310.482} C_VEL
LIN {X 0,Y 277.245,Z 420.95,A -85,B 0,C 180,E1 -17313.896,E2 -17313.896} C_VEL
LIN {X 0,Y 277.317,Z 421.075,A -85,B 0,C 180,E1 -17316.785,E2 -17316.785} C_VEL
LIN {X 0,Y 277.791,Z 424.067,A -85,B 0,C 180,E1 -17320.626,E2 -17320.626} C_VEL
LIN {X 0,Y 278.419,Z 427.842,A -85,B 0,C 180,E1 -17325.026,E2 -17325.026} C_VEL
LIN {X 0,Y 279.07,Z 431.697,A -85,B 0,C 180,E1 -17329.098,E2 -17329.098} C_VEL
LIN {X 0,Y 279.402,Z 435.63,A -85,B 0,C 180,E1 -17332.866,E2 -17332.866} C_VEL
LIN {X 0,Y 279.007,Z 439.432,A -85,B 0,C 180,E1 -17336.228,E2 -17336.228} C_VEL
LIN {X 0,Y 278.003,Z 444.778,A -85,B 0,C 180,E1 -17340.655,E2 -17340.655} C_VEL
LIN {X 0,Y 278.911,Z 448.031,A -85,B 0,C 180,E1 -17340.93,E2 -17340.93} C_VEL
LIN {X 0,Y 282.597,Z 459.615,A -85,B 0,C 180,E1 -17342.084,E2 -17342.084} C_VEL
LIN {X 0,Y 285.431,Z 471.089,A -85,B 0,C 180,E1 -17343.346,E2 -17343.346} C_VEL
LIN {X 0,Y 287.109,Z 481.42,A -85,B 0,C 180,E1 -17344.596,E2 -17344.596} C_VEL
LIN {X 0,Y 287.991,Z 492.273,A -85,B 0,C 180,E1 -17346.065,E2 -17346.065} C_VEL
LIN {X 0,Y 287.792,Z 498.725,A -85,B 0,C 180,E1 -17347,E2 -17347} C_VEL
LIN {X 0,Y 285.673,Z 507.65,A -85,B 0,C 180,E1 -17348.345,E2 -17348.345} C_VEL
LIN {X 0,Y 283.469,Z 516.828,A -85,B 0,C 180,E1 -17350.069,E2 -17350.069} C_VEL
LIN {X 0,Y 281.309,Z 525.926,A -85,B 0,C 180,E1 -17352.224,E2 -17352.224} C_VEL
LIN {X 0,Y 279.422,Z 532.999,A -85,B 0,C 180,E1 -17354.313,E2 -17354.313} C_VEL
LIN {X 0,Y 277.595,Z 539.648,A -85,B 0,C 180,E1 -17356.829,E2 -17356.829} C_VEL
LIN {X 0,Y 276.584,Z 544.066,A -85,B 0,C 180,E1 -17359.014,E2 -17359.014} C_VEL
LIN {X 0,Y 275.853,Z 547.433,A -85,B 0,C 180,E1 -17361.207,E2 -17361.207} C_VEL
LIN {X 0,Y 275.338,Z 550.411,A -85,B 0,C 180,E1 -17364.14,E2 -17364.14} C_VEL
LIN {X 0,Y 275.231,Z 551.315,A -85,B 0,C 180,E1 -17365.606,E2 -17365.606} C_VEL
LIN {X 0,Y 275.247,Z 551.797,A -85,B 0,C 180,E1 -17367.073,E2 -17367.073} C_VEL
LIN {X 0,Y 275.262,Z 551.877,A -85,B 0,C 180,E1 -17368.537,E2 -17368.537} C_VEL
LIN {X 0,Y 275.28,Z 551.572,A -85,B 0,C 180,E1 -17370,E2 -17370} C_VEL
LIN {X 0,Y 275.269,Z 550.879,A -85,B 0,C 180,E1 -17371.463,E2 -17371.463} C_VEL
LIN {X 0,Y 275.279,Z 549.76,A -85,B 0,C 180,E1 -17372.927,E2 -17372.927} C_VEL
LIN {X 0,Y 275.322,Z 546.867,A -85,B 0,C 180,E1 -17375.415,E2 -17375.415} C_VEL
LIN {X 0,Y 275.602,Z 542.355,A -85,B 0,C 180,E1 -17378.062,E2 -17378.062} C_VEL
LIN {X 0,Y 276.123,Z 537.349,A -85,B 0,C 180,E1 -17380.263,E2 -17380.263} C_VEL
LIN {X 0,Y 276.84,Z 531.035,A -85,B 0,C 180,E1 -17382.461,E2 -17382.461} C_VEL
LIN {X 0,Y 278.039,Z 523.126,A -85,B 0,C 180,E1 -17384.641,E2 -17384.641} C_VEL
LIN {X 0,Y 279.376,Z 514.024,A -85,B 0,C 180,E1 -17386.651,E2 -17386.651} C_VEL
LIN {X 0,Y 280.689,Z 504.06,A -85,B 0,C 180,E1 -17388.427,E2 -17388.427} C_VEL
LIN {X 0,Y 282.06,Z 494.101,A -85,B 0,C 180,E1 -17389.845,E2 -17389.845} C_VEL
LIN {X 0,Y 282.371,Z 489.736,A -85,B 0,C 180,E1 -17390.392,E2 -17390.392} C_VEL
LIN {X 0,Y 281.431,Z 477.92,A -85,B 0,C 180,E1 -17391.731,E2 -17391.731} C_VEL
LIN {X 0,Y 279.915,Z 465.242,A -85,B 0,C 180,E1 -17392.882,E2 -17392.882} C_VEL
LIN {X 0,Y 277.89,Z 452.729,A -85,B 0,C 180,E1 -17393.766,E2 -17393.766} C_VEL
LIN {X 0,Y 276.538,Z 445.446,A -85,B 0,C 180,E1 -17394.203,E2 -17394.203} C_VEL
LIN {X 0,Y 276.958,Z 441.216,A -85,B 0,C 180,E1 -17397.358,E2 -17397.358} C_VEL
LIN {X 0,Y 277.922,Z 434.98,A -85,B 0,C 180,E1 -17402.075,E2 -17402.075} C_VEL
LIN {X 0,Y 278.482,Z 430.638,A -85,B 0,C 180,E1 -17405.481,E2 -17405.481} C_VEL
LIN {X 0,Y 278.575,Z 428.434,A -85,B 0,C 180,E1 -17407.262,E2 -17407.262} C_VEL
LIN {X 0,Y 277.947,Z 424.474,A -85,B 0,C 180,E1 -17410.662,E2 -17410.662} C_VEL
LIN {X 0,Y 277.325,Z 420.941,A -85,B 0,C 180,E1 -17413.954,E2 -17413.954} C_VEL
LIN {X 0,Y 277.23,Z 420.955,A -85,B 0,C 180,E1 -17417.32,E2 -17417.32} C_VEL
LIN {X 0,Y 277.261,Z 420.947,A -85,B 0,C 180,E1 -17421.791,E2 -17421.791} C_VEL
LIN {X 0,Y 277.281,Z 420.945,A -85,B 0,C 180,E1 -17424.34,E2 -17424.34} C_VEL
LIN {X 0,Y 277.24,Z 420.948,A -85,B 0,C 180,E1 -17427.835,E2 -17427.835} C_VEL
LIN {X 0,Y 277.266,Z 420.94,A -85,B 0,C 180,E1 -17431.21,E2 -17431.21} C_VEL
LIN {X 0,Y 277.309,Z 420.938,A -85,B 0,C 180,E1 -17434.479,E2 -17434.479} C_VEL
LIN {X 0,Y 277.28,Z 420.943,A -85,B 0,C 180,E1 -17437.654,E2 -17437.654} C_VEL
LIN {X 0,Y 277.339,Z 420.934,A -85,B 0,C 180,E1 -17440.765,E2 -17440.765} C_VEL
LIN {X 0,Y 277.41,Z 420.922,A -85,B 0,C 180,E1 -17445.324,E2 -17445.324} C_VEL
LIN {X 0,Y 277.5,Z 420.916,A -85,B 0,C 180,E1 -17449.788,E2 -17449.788} C_VEL
LIN {X 0,Y 277.648,Z 420.896,A -85,B 0,C 180,E1 -17452.729,E2 -17452.729} C_VEL
LIN {X 0,Y 277.816,Z 420.872,A -85,B 0,C 180,E1 -17458.55,E2 -17458.55} C_VEL
LIN {X 0,Y 277.816,Z 420.875,A -85,B 0,C 180,E1 -17461.449,E2 -17461.449} C_VEL
LIN {X 0,Y 277.646,Z 420.895,A -85,B 0,C 180,E1 -17467.271,E2 -17467.271} C_VEL
LIN {X 0,Y 277.5,Z 420.907,A -85,B 0,C 180,E1 -17470.211,E2 -17470.211} C_VEL
LIN {X 0,Y 277.422,Z 420.923,A -85,B 0,C 180,E1 -17474.675,E2 -17474.675} C_VEL
LIN {X 0,Y 277.338,Z 420.936,A -85,B 0,C 180,E1 -17479.234,E2 -17479.234} C_VEL
LIN {X 0,Y 277.313,Z 420.942,A -85,B 0,C 180,E1 -17484.171,E2 -17484.171} C_VEL
LIN {X 0,Y 277.32,Z 420.94,A -85,B 0,C 180,E1 -17487.506,E2 -17487.506} C_VEL
LIN {X 0,Y 277.267,Z 420.945,A -85,B 0,C 180,E1 -17490.482,E2 -17490.482} C_VEL
LIN {X 0,Y 277.249,Z 420.949,A -85,B 0,C 180,E1 -17493.895,E2 -17493.895} C_VEL
LIN {X 0,Y 277.286,Z 420.944,A -85,B 0,C 180,E1 -17497.466,E2 -17497.466} C_VEL
LIN {X 0,Y 277.29,Z 420.943,A -85,B 0,C 180,E1 -17501.222,E2 -17501.222} C_VEL
LIN {X 0,Y 277.284,Z 420.945,A -85,B 0,C 180,E1 -17505.209,E2 -17505.209} C_VEL
LIN {X 0,Y 277.293,Z 420.946,A -85,B 0,C 180,E1 -17509.495,E2 -17509.495} C_VEL
LIN {X 0,Y 277.287,Z 420.943,A -85,B 0,C 180,E1 -17512.535,E2 -17512.535} C_VEL
LIN {X 0,Y 277.252,Z 420.947,A -85,B 0,C 180,E1 -17516.106,E2 -17516.106} C_VEL
LIN {X 0,Y 277.259,Z 420.949,A -85,B 0,C 180,E1 -17519.539,E2 -17519.539} C_VEL
LIN {X 0,Y 277.359,Z 420.936,A -85,B 0,C 180,E1 -17522.865,E2 -17522.865} C_VEL
LIN {X 0,Y 277.276,Z 420.945,A -85,B 0,C 180,E1 -17526.076,E2 -17526.076} C_VEL
LIN {X 0,Y 277.27,Z 420.984,A -85,B 0,C 180,E1 -17528.827,E2 -17528.827} C_VEL
LIN {X 0,Y 276.877,Z 424.179,A -85,B 0,C 180,E1 -17532.267,E2 -17532.267} C_VEL
LIN {X 0,Y 276.734,Z 427.057,A -85,B 0,C 180,E1 -17535.289,E2 -17535.289} C_VEL
LIN {X 0,Y 276.392,Z 431.666,A -85,B 0,C 180,E1 -17539.933,E2 -17539.933} C_VEL
LIN {X 0,Y 279.733,Z 444.905,A -85,B 0,C 180,E1 -17540.829,E2 -17540.829} C_VEL
LIN {X 0,Y 282.023,Z 457.307,A -85,B 0,C 180,E1 -17541.896,E2 -17541.896} C_VEL
LIN {X 0,Y 283.484,Z 468.278,A -85,B 0,C 180,E1 -17543.055,E2 -17543.055} C_VEL
LIN {X 0,Y 283.432,Z 472.06,A -85,B 0,C 180,E1 -17543.485,E2 -17543.485} C_VEL
LIN {X 0,Y 282.021,Z 483.488,A -85,B 0,C 180,E1 -17544.925,E2 -17544.925} C_VEL
LIN {X 0,Y 280.731,Z 492.883,A -85,B 0,C 180,E1 -17546.412,E2 -17546.412} C_VEL
LIN {X 0,Y 279.316,Z 502.048,A -85,B 0,C 180,E1 -17548.198,E2 -17548.198} C_VEL
LIN {X 0,Y 277.978,Z 510.967,A -85,B 0,C 180,E1 -17550.362,E2 -17550.362} C_VEL
LIN {X 0,Y 276.957,Z 518.137,A -85,B 0,C 180,E1 -17552.545,E2 -17552.545} C_VEL
LIN {X 0,Y 276.153,Z 524.657,A -85,B 0,C 180,E1 -17555.111,E2 -17555.111} C_VEL
LIN {X 0,Y 275.687,Z 528.974,A -85,B 0,C 180,E1 -17557.323,E2 -17557.323} C_VEL
LIN {X 0,Y 275.394,Z 531.274,A -85,B 0,C 180,E1 -17558.808,E2 -17558.808} C_VEL
LIN {X 0,Y 275.185,Z 533.104,A -85,B 0,C 180,E1 -17560.298,E2 -17560.298} C_VEL
LIN {X 0,Y 275.097,Z 534.479,A -85,B 0,C 180,E1 -17561.793,E2 -17561.793} C_VEL
LIN {X 0,Y 275.059,Z 535.714,A -85,B 0,C 180,E1 -17563.849,E2 -17563.849} C_VEL
LIN {X 0,Y 275.116,Z 536.149,A -85,B 0,C 180,E1 -17566.32,E2 -17566.32} C_VEL
LIN {X 0,Y 275.29,Z 535.859,A -85,B 0,C 180,E1 -17567.839,E2 -17567.839} C_VEL
LIN {X 0,Y 275.578,Z 535.166,A -85,B 0,C 180,E1 -17569.362,E2 -17569.362} C_VEL
LIN {X 0,Y 275.897,Z 534.025,A -85,B 0,C 180,E1 -17570.893,E2 -17570.893} C_VEL
LIN {X 0,Y 276.649,Z 531.465,A -85,B 0,C 180,E1 -17573.189,E2 -17573.189} C_VEL
LIN {X 0,Y 277.657,Z 527.807,A -85,B 0,C 180,E1 -17575.486,E2 -17575.486} C_VEL
LIN {X 0,Y 278.958,Z 523.206,A -85,B 0,C 180,E1 -17577.662,E2 -17577.662} C_VEL
LIN {X 0,Y 280.763,Z 516.69,A -85,B 0,C 180,E1 -17580.042,E2 -17580.042} C_VEL
LIN {X 0,Y 282.955,Z 508.465,A -85,B 0,C 180,E1 -17582.383,E2 -17582.383} C_VEL
LIN {X 0,Y 284.917,Z 500.703,A -85,B 0,C 180,E1 -17584.136,E2 -17584.136} C_VEL
LIN {X 0,Y 287.296,Z 490.671,A -85,B 0,C 180,E1 -17585.951,E2 -17585.951} C_VEL
LIN {X 0,Y 289.326,Z 480.763,A -85,B 0,C 180,E1 -17587.392,E2 -17587.392} C_VEL
LIN {X 0,Y 289.795,Z 476.606,A -85,B 0,C 180,E1 -17587.942,E2 -17587.942} C_VEL
LIN {X 0,Y 288.311,Z 467.003,A -85,B 0,C 180,E1 -17589.33,E2 -17589.33} C_VEL
LIN {X 0,Y 285.594,Z 455.592,A -85,B 0,C 180,E1 -17590.826,E2 -17590.826} C_VEL
LIN {X 0,Y 281.618,Z 443.487,A -85,B 0,C 180,E1 -17592.277,E2 -17592.277} C_VEL
LIN {X 0,Y 278.079,Z 435.09,A -85,B 0,C 180,E1 -17593.23,E2 -17593.23} C_VEL
LIN {X 0,Y 277.262,Z 432.319,A -85,B 0,C 180,E1 -17593.516,E2 -17593.516} C_VEL
LIN {X 0,Y 277.639,Z 429.198,A -85,B 0,C 180,E1 -17597.23,E2 -17597.23} C_VEL
LIN {X 0,Y 277.803,Z 426.416,A -85,B 0,C 180,E1 -17600.768,E2 -17600.768} C_VEL
LIN {X 0,Y 277.673,Z 423.76,A -85,B 0,C 180,E1 -17604.399,E2 -17604.399} C_VEL
LIN {X 0,Y 277.291,Z 421.454,A -85,B 0,C 180,E1 -17607.843,E2 -17607.843} C_VEL
LIN {X 0,Y 277.258,Z 420.95,A -85,B 0,C 180,E1 -17609.538,E2 -17609.538} C_VEL
LIN {X 0,Y 277.356,Z 420.938,A -85,B 0,C 180,E1 -17612.864,E2 -17612.864} C_VEL
LIN {X 0,Y 277.293,Z 420.943,A -85,B 0,C 180,E1 -17616.077,E2 -17616.077} C_VEL
LIN {X 0,Y 277.341,Z 420.936,A -85,B 0,C 180,E1 -17620.766,E2 -17620.766} C_VEL
LIN {X 0,Y 277.424,Z 420.926,A -85,B 0,C 180,E1 -17625.326,E2 -17625.326} C_VEL
LIN {X 0,Y 277.503,Z 420.915,A -85,B 0,C 180,E1 -17629.789,E2 -17629.789} C_VEL
LIN {X 0,Y 277.649,Z 420.901,A -85,B 0,C 180,E1 -17632.729,E2 -17632.729} C_VEL
LIN {X 0,Y 277.817,Z 420.879,A -85,B 0,C 180,E1 -17638.551,E2 -17638.551} C_VEL
LIN {X 0,Y 277.819,Z 420.88,A -85,B 0,C 180,E1 -17641.45,E2 -17641.45} C_VEL
LIN {X 0,Y 277.646,Z 420.893,A -85,B 0,C 180,E1 -17647.271,E2 -17647.271} C_VEL
LIN {X 0,Y 277.504,Z 420.918,A -85,B 0,C 180,E1 -17650.212,E2 -17650.212} C_VEL
LIN {X 0,Y 277.454,Z 420.922,A -85,B 0,C 180,E1 -17650.795,E2 -17650.795} C_VEL
LIN {X 0,Y 276.745,Z 421.013,A -85,B 0,C 180,E1 -17652.007,E2 -17652.007} C_VEL
LIN {X 0,Y 273.884,Z 421.369,A -85,B 0,C 180,E1 -17653.982,E2 -17653.982} C_VEL
LIN {X 0,Y 271.464,Z 421.671,A -85,B 0,C 180,E1 -17655.586,E2 -17655.586} C_VEL
LIN {X 0,Y 270.402,Z 421.805,A -85,B 0,C 180,E1 -17656.83,E2 -17656.83} C_VEL
LIN {X 0,Y 270.302,Z 421.815,A -85,B 0,C 180,E1 -17657.251,E2 -17657.251} C_VEL
LIN {X 0,Y 270.29,Z 421.82,A -85,B 0,C 180,E1 -17660.602,E2 -17660.602} C_VEL
LIN {X 0,Y 270.272,Z 421.823,A -85,B 0,C 180,E1 -17664.586,E2 -17664.586} C_VEL
LIN {X 0,Y 270.27,Z 421.822,A -85,B 0,C 180,E1 -17667.909,E2 -17667.909} C_VEL
LIN {X 0,Y 270.183,Z 421.83,A -85,B 0,C 180,E1 -17671.349,E2 -17671.349} C_VEL
LIN {X 0,Y 270.246,Z 421.857,A -85,B 0,C 180,E1 -17675.689,E2 -17675.689} C_VEL
LIN {X 0,Y 270.643,Z 424.135,A -85,B 0,C 180,E1 -17678.829,E2 -17678.829} C_VEL
LIN {X 0,Y 271.05,Z 426.982,A -85,B 0,C 180,E1 -17682.389,E2 -17682.389} C_VEL
LIN {X 0,Y 271.671,Z 430.481,A -85,B 0,C 180,E1 -17686.415,E2 -17686.415} C_VEL
LIN {X 0,Y 272.144,Z 433.674,A -85,B 0,C 180,E1 -17689.789,E2 -17689.789} C_VEL
LIN {X 0,Y 272.399,Z 437.072,A -85,B 0,C 180,E1 -17693.113,E2 -17693.113} C_VEL
LIN {X 0,Y 272.047,Z 439.994,A -85,B 0,C 180,E1 -17695.76,E2 -17695.76} C_VEL
LIN {X 0,Y 271.159,Z 444.572,A -85,B 0,C 180,E1 -17699.671,E2 -17699.671} C_VEL
LIN {X 0,Y 272.054,Z 447.739,A -85,B 0,C 180,E1 -17699.947,E2 -17699.947} C_VEL
LIN {X 0,Y 275.975,Z 459.652,A -85,B 0,C 180,E1 -17701.21,E2 -17701.21} C_VEL
LIN {X 0,Y 278.972,Z 471.888,A -85,B 0,C 180,E1 -17702.628,E2 -17702.628} C_VEL
LIN {X 0,Y 280.744,Z 483.244,A -85,B 0,C 180,E1 -17704.079,E2 -17704.079} C_VEL
LIN {X 0,Y 281.439,Z 493.022,A -85,B 0,C 180,E1 -17705.471,E2 -17705.471} C_VEL
LIN {X 0,Y 281.287,Z 499.314,A -85,B 0,C 180,E1 -17706.437,E2 -17706.437} C_VEL
LIN {X 0,Y 279.103,Z 508.109,A -85,B 0,C 180,E1 -17707.808,E2 -17707.808} C_VEL
LIN {X 0,Y 276.815,Z 517.16,A -85,B 0,C 180,E1 -17709.568,E2 -17709.568} C_VEL
LIN {X 0,Y 274.523,Z 526.275,A -85,B 0,C 180,E1 -17711.801,E2 -17711.801} C_VEL
LIN {X 0,Y 272.6,Z 533.153,A -85,B 0,C 180,E1 -17713.91,E2 -17713.91} C_VEL
LIN {X 0,Y 270.66,Z 539.699,A -85,B 0,C 180,E1 -17716.485,E2 -17716.485} C_VEL
LIN {X 0,Y 269.594,Z 544.056,A -85,B 0,C 180,E1 -17718.725,E2 -17718.725} C_VEL
LIN {X 0,Y 268.825,Z 547.368,A -85,B 0,C 180,E1 -17720.975,E2 -17720.975} C_VEL
LIN {X 0,Y 268.25,Z 550.294,A -85,B 0,C 180,E1 -17723.984,E2 -17723.984} C_VEL
LIN {X 0,Y 268.151,Z 551.163,A -85,B 0,C 180,E1 -17725.49,E2 -17725.49} C_VEL
LIN {X 0,Y 268.159,Z 551.605,A -85,B 0,C 180,E1 -17726.995,E2 -17726.995} C_VEL
LIN {X 0,Y 268.187,Z 551.66,A -85,B 0,C 180,E1 -17728.498,E2 -17728.498} C_VEL
LIN {X 0,Y 268.203,Z 551.33,A -85,B 0,C 180,E1 -17730,E2 -17730} C_VEL
LIN {X 0,Y 268.196,Z 550.609,A -85,B 0,C 180,E1 -17731.501,E2 -17731.501} C_VEL
LIN {X 0,Y 268.189,Z 549.441,A -85,B 0,C 180,E1 -17733.004,E2 -17733.004} C_VEL
LIN {X 0,Y 268.214,Z 546.855,A -85,B 0,C 180,E1 -17735.304,E2 -17735.304} C_VEL
LIN {X 0,Y 268.417,Z 543.362,A -85,B 0,C 180,E1 -17737.522,E2 -17737.522} C_VEL
LIN {X 0,Y 268.888,Z 538.685,A -85,B 0,C 180,E1 -17739.781,E2 -17739.781} C_VEL
LIN {X 0,Y 269.702,Z 531.603,A -85,B 0,C 180,E1 -17742.414,E2 -17742.414} C_VEL
LIN {X 0,Y 270.922,Z 523.936,A -85,B 0,C 180,E1 -17744.65,E2 -17744.65} C_VEL
LIN {X 0,Y 272.32,Z 514.865,A -85,B 0,C 180,E1 -17746.75,E2 -17746.75} C_VEL
LIN {X 0,Y 273.584,Z 505.334,A -85,B 0,C 180,E1 -17748.535,E2 -17748.535} C_VEL
LIN {X 0,Y 274.911,Z 495.713,A -85,B 0,C 180,E1 -17749.994,E2 -17749.994} C_VEL
LIN {X 0,Y 275.487,Z 491.542,A -85,B 0,C 180,E1 -17750.534,E2 -17750.534} C_VEL
LIN {X 0,Y 274.665,Z 479.762,A -85,B 0,C 180,E1 -17751.968,E2 -17751.968} C_VEL
LIN {X 0,Y 273.419,Z 468.46,A -85,B 0,C 180,E1 -17753.077,E2 -17753.077} C_VEL
LIN {X 0,Y 271.548,Z 455.964,A -85,B 0,C 180,E1 -17754.045,E2 -17754.045} C_VEL
LIN {X 0,Y 269.546,Z 445.292,A -85,B 0,C 180,E1 -17754.707,E2 -17754.707} C_VEL
LIN {X 0,Y 270.237,Z 438.917,A -85,B 0,C 180,E1 -17759.611,E2 -17759.611} C_VEL
LIN {X 0,Y 271.004,Z 434.607,A -85,B 0,C 180,E1 -17762.996,E2 -17762.996} C_VEL
LIN {X 0,Y 271.469,Z 431.345,A -85,B 0,C 180,E1 -17765.625,E2 -17765.625} C_VEL
LIN {X 0,Y 271.506,Z 429.146,A -85,B 0,C 180,E1 -17767.465,E2 -17767.465} C_VEL
LIN {X 0,Y 270.989,Z 425.8,A -85,B 0,C 180,E1 -17770.417,E2 -17770.417} C_VEL
LIN {X 0,Y 270.271,Z 421.82,A -85,B 0,C 180,E1 -17774.191,E2 -17774.191} C_VEL
LIN {X 0,Y 270.184,Z 421.832,A -85,B 0,C 180,E1 -17777.444,E2 -17777.444} C_VEL
LIN {X 0,Y 270.204,Z 421.829,A -85,B 0,C 180,E1 -17781.373,E2 -17781.373} C_VEL
LIN {X 0,Y 270.198,Z 421.83,A -85,B 0,C 180,E1 -17785.094,E2 -17785.094} C_VEL
LIN {X 0,Y 270.196,Z 421.827,A -85,B 0,C 180,E1 -17789.13,E2 -17789.13} C_VEL
LIN {X 0,Y 270.259,Z 421.811,A -85,B 0,C 180,E1 -17792.145,E2 -17792.145} C_VEL
LIN {X 0,Y 270.272,Z 421.816,A -85,B 0,C 180,E1 -17795.518,E2 -17795.518} C_VEL
LIN {X 0,Y 270.296,Z 421.813,A -85,B 0,C 180,E1 -17800.244,E2 -17800.244} C_VEL
LIN {X 0,Y 270.377,Z 421.8,A -85,B 0,C 180,E1 -17804.934,E2 -17804.934} C_VEL
LIN {X 0,Y 270.436,Z 421.796,A -85,B 0,C 180,E1 -17809.518,E2 -17809.518} C_VEL
LIN {X 0,Y 270.606,Z 421.775,A -85,B 0,C 180,E1 -17812.538,E2 -17812.538} C_VEL
LIN {X 0,Y 270.782,Z 421.746,A -85,B 0,C 180,E1 -17818.512,E2 -17818.512} C_VEL
LIN {X 0,Y 270.782,Z 421.751,A -85,B 0,C 180,E1 -17821.487,E2 -17821.487} C_VEL
LIN {X 0,Y 270.605,Z 421.772,A -85,B 0,C 180,E1 -17827.461,E2 -17827.461} C_VEL
LIN {X 0,Y 270.435,Z 421.783,A -85,B 0,C 180,E1 -17830.481,E2 -17830.481} C_VEL
LIN {X 0,Y 270.39,Z 421.798,A -85,B 0,C 180,E1 -17835.065,E2 -17835.065} C_VEL
LIN {X 0,Y 270.295,Z 421.816,A -85,B 0,C 180,E1 -17839.756,E2 -17839.756} C_VEL
LIN {X 0,Y 270.268,Z 421.817,A -85,B 0,C 180,E1 -17844.586,E2 -17844.586} C_VEL
LIN {X 0,Y 270.265,Z 421.818,A -85,B 0,C 180,E1 -17847.909,E2 -17847.909} C_VEL
LIN {X 0,Y 270.18,Z 421.829,A -85,B 0,C 180,E1 -17851.349,E2 -17851.349} C_VEL
LIN {X 0,Y 270.211,Z 421.822,A -85,B 0,C 180,E1 -17854.904,E2 -17854.904} C_VEL
LIN {X 0,Y 270.218,Z 421.823,A -85,B 0,C 180,E1 -17858.718,E2 -17858.718} C_VEL
LIN {X 0,Y 270.253,Z 421.819,A -85,B 0,C 180,E1 -17862.542,E2 -17862.542} C_VEL
LIN {X 0,Y 270.231,Z 421.821,A -85,B 0,C 180,E1 -17866.736,E2 -17866.736} C_VEL
LIN {X 0,Y 270.246,Z 421.823,A -85,B 0,C 180,E1 -17869.449,E2 -17869.449} C_VEL
LIN {X 0,Y 270.255,Z 421.82,A -85,B 0,C 180,E1 -17873.722,E2 -17873.722} C_VEL
LIN {X 0,Y 270.202,Z 421.826,A -85,B 0,C 180,E1 -17876.893,E2 -17876.893} C_VEL
LIN {X 0,Y 270.227,Z 421.822,A -85,B 0,C 180,E1 -17880.387,E2 -17880.387} C_VEL
LIN {X 0,Y 270.258,Z 421.82,A -85,B 0,C 180,E1 -17883.764,E2 -17883.764} C_VEL
LIN {X 0,Y 270.265,Z 421.822,A -85,B 0,C 180,E1 -17888.715,E2 -17888.715} C_VEL
LIN {X 0,Y 269.745,Z 426.03,A -85,B 0,C 180,E1 -17893.346,E2 -17893.346} C_VEL
LIN {X 0,Y 269.55,Z 428.928,A -85,B 0,C 180,E1 -17896.429,E2 -17896.429} C_VEL
LIN {X 0,Y 269.343,Z 431.778,A -85,B 0,C 180,E1 -17899.381,E2 -17899.381} C_VEL
LIN {X 0,Y 273.103,Z 446.677,A -85,B 0,C 180,E1 -17900.464,E2 -17900.464} C_VEL
LIN {X 0,Y 275.269,Z 458.801,A -85,B 0,C 180,E1 -17901.56,E2 -17901.56} C_VEL
LIN {X 0,Y 276.759,Z 470.59,A -85,B 0,C 180,E1 -17902.885,E2 -17902.885} C_VEL
LIN {X 0,Y 275.412,Z 481.934,A -85,B 0,C 180,E1 -17904.307,E2 -17904.307} C_VEL
LIN {X 0,Y 273.9,Z 492.416,A -85,B 0,C 180,E1 -17905.954,E2 -17905.954} C_VEL
LIN {X 0,Y 272.477,Z 501.709,A -85,B 0,C 180,E1 -17907.783,E2 -17907.783} C_VEL
LIN {X 0,Y 271.056,Z 510.721,A -85,B 0,C 180,E1 -17910,E2 -17910} C_VEL
LIN {X 0,Y 269.961,Z 517.982,A -85,B 0,C 180,E1 -17912.238,E2 -17912.238} C_VEL
LIN {X 0,Y 269.175,Z 523.782,A -85,B 0,C 180,E1 -17914.493,E2 -17914.493} C_VEL
LIN {X 0,Y 268.75,Z 527.722,A -85,B 0,C 180,E1 -17916.422,E2 -17916.422} C_VEL
LIN {X 0,Y 268.274,Z 531.824,A -85,B 0,C 180,E1 -17919.044,E2 -17919.044} C_VEL
LIN {X 0,Y 268.056,Z 533.559,A -85,B 0,C 180,E1 -17920.575,E2 -17920.575} C_VEL
LIN {X 0,Y 268.009,Z 534.878,A -85,B 0,C 180,E1 -17922.11,E2 -17922.11} C_VEL
LIN {X 0,Y 267.969,Z 535.924,A -85,B 0,C 180,E1 -17923.977,E2 -17923.977} C_VEL
LIN {X 0,Y 268.051,Z 536.331,A -85,B 0,C 180,E1 -17926.763,E2 -17926.763} C_VEL
LIN {X 0,Y 268.53,Z 535.396,A -85,B 0,C 180,E1 -17929.577,E2 -17929.577} C_VEL
LIN {X 0,Y 268.958,Z 533.981,A -85,B 0,C 180,E1 -17931.458,E2 -17931.458} C_VEL
LIN {X 0,Y 270.038,Z 530.526,A -85,B 0,C 180,E1 -17934.369,E2 -17934.369} C_VEL
LIN {X 0,Y 271.397,Z 526.016,A -85,B 0,C 180,E1 -17936.947,E2 -17936.947} C_VEL
LIN {X 0,Y 273.294,Z 519.507,A -85,B 0,C 180,E1 -17939.671,E2 -17939.671} C_VEL
LIN {X 0,Y 275.426,Z 512.345,A -85,B 0,C 180,E1 -17941.969,E2 -17941.969} C_VEL
LIN {X 0,Y 277.415,Z 504.925,A -85,B 0,C 180,E1 -17943.872,E2 -17943.872} C_VEL
LIN {X 0,Y 279.742,Z 495.842,A -85,B 0,C 180,E1 -17945.74,E2 -17945.74} C_VEL
LIN {X 0,Y 282.221,Z 485.054,A -85,B 0,C 180,E1 -17947.507,E2 -17947.507} C_VEL
LIN {X 0,Y 283.389,Z 479.143,A -85,B 0,C 180,E1 -17948.315,E2 -17948.315} C_VEL
LIN {X 0,Y 282.419,Z 471.307,A -85,B 0,C 180,E1 -17949.517,E2 -17949.517} C_VEL
LIN {X 0,Y 279.965,Z 459.928,A -85,B 0,C 180,E1 -17951.141,E2 -17951.141} C_VEL
LIN {X 0,Y 276.564,Z 448.591,A -85,B 0,C 180,E1 -17952.61,E2 -17952.61} C_VEL
LIN {X 0,Y 271.844,Z 436.437,A -85,B 0,C 180,E1 -17954.069,E2 -17954.069} C_VEL
LIN {X 0,Y 270.442,Z 433.255,A -85,B 0,C 180,E1 -17954.44,E2 -17954.44} C_VEL
LIN {X 0,Y 270.348,Z 432.554,A -85,B 0,C 180,E1 -17954.531,E2 -17954.531} C_VEL
LIN {X 0,Y 270.647,Z 430.117,A -85,B 0,C 180,E1 -17957.534,E2 -17957.534} C_VEL
LIN {X 0,Y 270.796,Z 428.539,A -85,B 0,C 180,E1 -17959.547,E2 -17959.547} C_VEL
LIN {X 0,Y 270.73,Z 425.781,A -85,B 0,C 180,E1 -17963.34,E2 -17963.34} C_VEL
LIN {X 0,Y 270.428,Z 423.382,A -85,B 0,C 180,E1 -17966.924,E2 -17966.924} C_VEL
LIN {X 0,Y 270.243,Z 422.007,A -85,B 0,C 180,E1 -17969.114,E2 -17969.114} C_VEL
LIN {X 0,Y 270.262,Z 421.82,A -85,B 0,C 180,E1 -17972.145,E2 -17972.145} C_VEL
LIN {X 0,Y 270.234,Z 421.823,A -85,B 0,C 180,E1 -17975.538,E2 -17975.538} C_VEL
LIN {X 0,Y 270.298,Z 421.813,A -85,B 0,C 180,E1 -17980.244,E2 -17980.244} C_VEL
LIN {X 0,Y 270.393,Z 421.803,A -85,B 0,C 180,E1 -17984.935,E2 -17984.935} C_VEL
LIN {X 0,Y 270.438,Z 421.793,A -85,B 0,C 180,E1 -17989.519,E2 -17989.519} C_VEL
LIN {X 0,Y 270.607,Z 421.778,A -85,B 0,C 180,E1 -17992.539,E2 -17992.539} C_VEL
LIN {X 0,Y 270.783,Z 421.755,A -85,B 0,C 180,E1 -17998.513,E2 -17998.513} C_VEL
LIN {X 0,Y 270.784,Z 421.756,A -85,B 0,C 180,E1 -18001.487,E2 -18001.487} C_VEL
LIN {X 0,Y 270.604,Z 421.77,A -85,B 0,C 180,E1 -18007.462,E2 -18007.462} C_VEL
LIN {X 0,Y 270.416,Z 421.799,A -85,B 0,C 180,E1 -18010.775,E2 -18010.775} C_VEL
LIN {X 0,Y 270.4,Z 421.804,A -85,B 0,C 180,E1 -18015.065,E2 -18015.065} C_VEL
LIN {X 0,Y 270.302,Z 421.815,A -85,B 0,C 180,E1 -18017.251,E2 -18017.251} C_VEL
LIN {X 0,Y 269.588,Z 421.908,A -85,B 0,C 180,E1 -18018.494,E2 -18018.494} C_VEL
LIN {X 0,Y 266.7,Z 422.267,A -85,B 0,C 180,E1 -18020.519,E2 -18020.519} C_VEL
LIN {X 0,Y 264.282,Z 422.569,A -85,B 0,C 180,E1 -18022.166,E2 -18022.166} C_VEL
LIN {X 0,Y 263.259,Z 422.696,A -85,B 0,C 180,E1 -18023.442,E2 -18023.442} C_VEL
LIN {X 0,Y 263.181,Z 422.704,A -85,B 0,C 180,E1 -18023.875,E2 -18023.875} C_VEL
LIN {X 0,Y 263.199,Z 422.702,A -85,B 0,C 180,E1 -18028.217,E2 -18028.217} C_VEL
LIN {X 0,Y 263.131,Z 422.709,A -85,B 0,C 180,E1 -18032.289,E2 -18032.289} C_VEL
LIN {X 0,Y 263.15,Z 422.705,A -85,B 0,C 180,E1 -18034.115,E2 -18034.115} C_VEL
LIN {X 0,Y 263.473,Z 424.207,A -85,B 0,C 180,E1 -18036.849,E2 -18036.849} C_VEL
LIN {X 0,Y 263.784,Z 426.344,A -85,B 0,C 180,E1 -18039.75,E2 -18039.75} C_VEL
LIN {X 0,Y 264.338,Z 429.851,A -85,B 0,C 180,E1 -18044.123,E2 -18044.123} C_VEL
LIN {X 0,Y 264.918,Z 433.244,A -85,B 0,C 180,E1 -18047.972,E2 -18047.972} C_VEL
LIN {X 0,Y 265.222,Z 435.651,A -85,B 0,C 180,E1 -18050.509,E2 -18050.509} C_VEL
LIN {X 0,Y 265.353,Z 437.736,A -85,B 0,C 180,E1 -18052.615,E2 -18052.615} C_VEL
LIN {X 0,Y 265.088,Z 440.564,A -85,B 0,C 180,E1 -18055.273,E2 -18055.273} C_VEL
LIN {X 0,Y 264.363,Z 444.309,A -85,B 0,C 180,E1 -18058.603,E2 -18058.603} C_VEL
LIN {X 0,Y 265.293,Z 447.648,A -85,B 0,C 180,E1 -18058.922,E2 -18058.922} C_VEL
LIN {X 0,Y 268.762,Z 457.833,A -85,B 0,C 180,E1 -18060.059,E2 -18060.059} C_VEL
LIN {X 0,Y 271.897,Z 469.83,A -85,B 0,C 180,E1 -18061.502,E2 -18061.502} C_VEL
LIN {X 0,Y 273.944,Z 481.171,A -85,B 0,C 180,E1 -18063.004,E2 -18063.004} C_VEL
LIN {X 0,Y 274.883,Z 492.437,A -85,B 0,C 180,E1 -18064.649,E2 -18064.649} C_VEL
LIN {X 0,Y 274.797,Z 499.888,A -85,B 0,C 180,E1 -18065.845,E2 -18065.845} C_VEL
LIN {X 0,Y 272.08,Z 510.484,A -85,B 0,C 180,E1 -18067.604,E2 -18067.604} C_VEL
LIN {X 0,Y 269.76,Z 519.111,A -85,B 0,C 180,E1 -18069.408,E2 -18069.408} C_VEL
LIN {X 0,Y 267.476,Z 527.521,A -85,B 0,C 180,E1 -18071.621,E2 -18071.621} C_VEL
LIN {X 0,Y 265.453,Z 534.307,A -85,B 0,C 180,E1 -18073.86,E2 -18073.86} C_VEL
LIN {X 0,Y 263.737,Z 539.762,A -85,B 0,C 180,E1 -18076.124,E2 -18076.124} C_VEL
LIN {X 0,Y 262.618,Z 544.056,A -85,B 0,C 180,E1 -18078.421,E2 -18078.421} C_VEL
LIN {X 0,Y 261.788,Z 547.309,A -85,B 0,C 180,E1 -18080.73,E2 -18080.73} C_VEL
LIN {X 0,Y 261.17,Z 550.179,A -85,B 0,C 180,E1 -18083.821,E2 -18083.821} C_VEL
LIN {X 0,Y 261.068,Z 551,A -85,B 0,C 180,E1 -18085.368,E2 -18085.368} C_VEL
LIN {X 0,Y 261.074,Z 551.413,A -85,B 0,C 180,E1 -18086.914,E2 -18086.914} C_VEL
LIN {X 0,Y 261.114,Z 551.444,A -85,B 0,C 180,E1 -18088.457,E2 -18088.457} C_VEL
LIN {X 0,Y 261.129,Z 551.089,A -85,B 0,C 180,E1 -18090,E2 -18090} C_VEL
LIN {X 0,Y 261.123,Z 550.327,A -85,B 0,C 180,E1 -18091.542,E2 -18091.542} C_VEL
LIN {X 0,Y 261.102,Z 549.122,A -85,B 0,C 180,E1 -18093.086,E2 -18093.086} C_VEL
LIN {X 0,Y 261.125,Z 546.784,A -85,B 0,C 180,E1 -18095.23,E2 -18095.23} C_VEL
LIN {X 0,Y 261.351,Z 542.93,A -85,B 0,C 180,E1 -18097.727,E2 -18097.727} C_VEL
LIN {X 0,Y 261.842,Z 538.19,A -85,B 0,C 180,E1 -18100.047,E2 -18100.047} C_VEL
LIN {X 0,Y 262.731,Z 531.041,A -85,B 0,C 180,E1 -18102.749,E2 -18102.749} C_VEL
LIN {X 0,Y 263.996,Z 523.266,A -85,B 0,C 180,E1 -18105.043,E2 -18105.043} C_VEL
LIN {X 0,Y 265.455,Z 513.867,A -85,B 0,C 180,E1 -18107.242,E2 -18107.242} C_VEL
LIN {X 0,Y 266.814,Z 504.434,A -85,B 0,C 180,E1 -18109.023,E2 -18109.023} C_VEL
LIN {X 0,Y 268.256,Z 494.673,A -85,B 0,C 180,E1 -18110.512,E2 -18110.512} C_VEL
LIN {X 0,Y 268.484,Z 490.348,A -85,B 0,C 180,E1 -18111.095,E2 -18111.095} C_VEL
LIN {X 0,Y 267.658,Z 478.998,A -85,B 0,C 180,E1 -18112.493,E2 -18112.493} C_VEL
LIN {X 0,Y 266.321,Z 467.01,A -85,B 0,C 180,E1 -18113.679,E2 -18113.679} C_VEL
LIN {X 0,Y 264.326,Z 454.442,A -85,B 0,C 180,E1 -18114.666,E2 -18114.666} C_VEL
LIN {X 0,Y 262.517,Z 445.1,A -85,B 0,C 180,E1 -18115.259,E2 -18115.259} C_VEL
LIN {X 0,Y 263.177,Z 439.62,A -85,B 0,C 180,E1 -18119.605,E2 -18119.605} C_VEL
LIN {X 0,Y 263.953,Z 435.296,A -85,B 0,C 180,E1 -18123.08,E2 -18123.08} C_VEL
LIN {X 0,Y 264.446,Z 432.051,A -85,B 0,C 180,E1 -18125.779,E2 -18125.779} C_VEL
LIN {X 0,Y 264.35,Z 428.843,A -85,B 0,C 180,E1 -18128.579,E2 -18128.579} C_VEL
LIN {X 0,Y 263.528,Z 424.227,A -85,B 0,C 180,E1 -18132.851,E2 -18132.851} C_VEL
LIN {X 0,Y 263.197,Z 422.702,A -85,B 0,C 180,E1 -18134.453,E2 -18134.453} C_VEL
LIN {X 0,Y 263.127,Z 422.71,A -85,B 0,C 180,E1 -18138.404,E2 -18138.404} C_VEL
LIN {X 0,Y 263.179,Z 422.704,A -85,B 0,C 180,E1 -18143.236,E2 -18143.236} C_VEL
LIN {X 0,Y 263.129,Z 422.707,A -85,B 0,C 180,E1 -18147.711,E2 -18147.711} C_VEL
LIN {X 0,Y 263.195,Z 422.69,A -85,B 0,C 180,E1 -18151.783,E2 -18151.783} C_VEL
LIN {X 0,Y 263.221,Z 422.695,A -85,B 0,C 180,E1 -18155.2,E2 -18155.2} C_VEL
LIN {X 0,Y 263.258,Z 422.688,A -85,B 0,C 180,E1 -18159.693,E2 -18159.693} C_VEL
LIN {X 0,Y 263.323,Z 422.671,A -85,B 0,C 180,E1 -18164.52,E2 -18164.52} C_VEL
LIN {X 0,Y 263.368,Z 422.677,A -85,B 0,C 180,E1 -18169.234,E2 -18169.234} C_VEL
LIN {X 0,Y 263.568,Z 422.653,A -85,B 0,C 180,E1 -18172.338,E2 -18172.338} C_VEL
LIN {X 0,Y 263.746,Z 422.62,A -85,B 0,C 180,E1 -18178.473,E2 -18178.473} C_VEL
LIN {X 0,Y 263.746,Z 422.627,A -85,B 0,C 180,E1 -18181.527,E2 -18181.527} C_VEL
LIN {X 0,Y 263.566,Z 422.649,A -85,B 0,C 180,E1 -18187.662,E2 -18187.662} C_VEL
LIN {X 0,Y 263.368,Z 422.66,A -85,B 0,C 180,E1 -18190.766,E2 -18190.766} C_VEL
LIN {X 0,Y 263.339,Z 422.677,A -85,B 0,C 180,E1 -18195.478,E2 -18195.478} C_VEL
LIN {X 0,Y 263.258,Z 422.69,A -85,B 0,C 180,E1 -18200.307,E2 -18200.307} C_VEL
LIN {X 0,Y 263.203,Z 422.698,A -85,B 0,C 180,E1 -18205.292,E2 -18205.292} C_VEL
LIN {X 0,Y 263.161,Z 422.698,A -85,B 0,C 180,E1 -18208.731,E2 -18208.731} C_VEL
LIN {X 0,Y 263.129,Z 422.707,A -85,B 0,C 180,E1 -18212.289,E2 -18212.289} C_VEL
LIN {X 0,Y 263.186,Z 422.7,A -85,B 0,C 180,E1 -18215.978,E2 -18215.978} C_VEL
LIN {X 0,Y 263.158,Z 422.705,A -85,B 0,C 180,E1 -18219.863,E2 -18219.863} C_VEL
LIN {X 0,Y 263.187,Z 422.701,A -85,B 0,C 180,E1 -18223.865,E2 -18223.865} C_VEL
LIN {X 0,Y 263.211,Z 422.696,A -85,B 0,C 180,E1 -18228.385,E2 -18228.385} C_VEL
LIN {X 0,Y 263.203,Z 422.7,A -85,B 0,C 180,E1 -18233.231,E2 -18233.231} C_VEL
LIN {X 0,Y 263.181,Z 422.701,A -85,B 0,C 180,E1 -18235.891,E2 -18235.891} C_VEL
LIN {X 0,Y 263.149,Z 422.707,A -85,B 0,C 180,E1 -18239.508,E2 -18239.508} C_VEL
LIN {X 0,Y 263.19,Z 422.702,A -85,B 0,C 180,E1 -18243.003,E2 -18243.003} C_VEL
LIN {X 0,Y 263.138,Z 422.707,A -85,B 0,C 180,E1 -18246.383,E2 -18246.383} C_VEL
LIN {X 0,Y 263.223,Z 422.704,A -85,B 0,C 180,E1 -18248.636,E2 -18248.636} C_VEL
LIN {X 0,Y 262.726,Z 426.493,A -85,B 0,C 180,E1 -18252.888,E2 -18252.888} C_VEL
LIN {X 0,Y 262.516,Z 429.38,A -85,B 0,C 180,E1 -18256.058,E2 -18256.058} C_VEL
LIN {X 0,Y 262.299,Z 431.98,A -85,B 0,C 180,E1 -18258.83,E2 -18258.83} C_VEL
LIN {X 0,Y 265.87,Z 445.855,A -85,B 0,C 180,E1 -18259.861,E2 -18259.861} C_VEL
LIN {X 0,Y 268.095,Z 457.687,A -85,B 0,C 180,E1 -18260.951,E2 -18260.951} C_VEL
LIN {X 0,Y 269.751,Z 470.008,A -85,B 0,C 180,E1 -18262.346,E2 -18262.346} C_VEL
LIN {X 0,Y 269.674,Z 473.687,A -85,B 0,C 180,E1 -18262.797,E2 -18262.797} C_VEL
LIN {X 0,Y 268.158,Z 485.148,A -85,B 0,C 180,E1 -18264.36,E2 -18264.36} C_VEL
LIN {X 0,Y 266.518,Z 495.891,A -85,B 0,C 180,E1 -18266.22,E2 -18266.22} C_VEL
LIN {X 0,Y 265.085,Z 504.625,A -85,B 0,C 180,E1 -18268.101,E2 -18268.101} C_VEL
LIN {X 0,Y 263.671,Z 513.103,A -85,B 0,C 180,E1 -18270.382,E2 -18270.382} C_VEL
LIN {X 0,Y 262.683,Z 519.901,A -85,B 0,C 180,E1 -18272.684,E2 -18272.684} C_VEL
LIN {X 0,Y 261.902,Z 526.149,A -85,B 0,C 180,E1 -18275.389,E2 -18275.389} C_VEL
LIN {X 0,Y 261.391,Z 530.225,A -85,B 0,C 180,E1 -18277.726,E2 -18277.726} C_VEL
LIN {X 0,Y 261.138,Z 532.333,A -85,B 0,C 180,E1 -18279.293,E2 -18279.293} C_VEL
LIN {X 0,Y 260.935,Z 534.011,A -85,B 0,C 180,E1 -18280.868,E2 -18280.868} C_VEL
LIN {X 0,Y 260.886,Z 535.277,A -85,B 0,C 180,E1 -18282.446,E2 -18282.446} C_VEL
LIN {X 0,Y 260.88,Z 536.133,A -85,B 0,C 180,E1 -18284.112,E2 -18284.112} C_VEL
LIN {X 0,Y 260.999,Z 536.513,A -85,B 0,C 180,E1 -18287.229,E2 -18287.229} C_VEL
LIN {X 0,Y 261.478,Z 535.618,A -85,B 0,C 180,E1 -18289.826,E2 -18289.826} C_VEL
LIN {X 0,Y 262.051,Z 533.943,A -85,B 0,C 180,E1 -18292.053,E2 -18292.053} C_VEL
LIN {X 0,Y 263.089,Z 530.79,A -85,B 0,C 180,E1 -18294.735,E2 -18294.735} C_VEL
LIN {X 0,Y 264.244,Z 527.242,A -85,B 0,C 180,E1 -18296.881,E2 -18296.881} C_VEL
LIN {X 0,Y 266.096,Z 521.374,A -85,B 0,C 180,E1 -18299.577,E2 -18299.577} C_VEL
LIN {X 0,Y 268.277,Z 514.271,A -85,B 0,C 180,E1 -18302.038,E2 -18302.038} C_VEL
LIN {X 0,Y 270.782,Z 505.704,A -85,B 0,C 180,E1 -18304.363,E2 -18304.363} C_VEL
LIN {X 0,Y 273.195,Z 496.744,A -85,B 0,C 180,E1 -18306.276,E2 -18306.276} C_VEL
LIN {X 0,Y 275.594,Z 486.834,A -85,B 0,C 180,E1 -18307.967,E2 -18307.967} C_VEL
LIN {X 0,Y 276.915,Z 480.301,A -85,B 0,C 180,E1 -18308.913,E2 -18308.913} C_VEL
LIN {X 0,Y 275.686,Z 471.122,A -85,B 0,C 180,E1 -18310.395,E2 -18310.395} C_VEL
LIN {X 0,Y 273.494,Z 460.805,A -85,B 0,C 180,E1 -18311.922,E2 -18311.922} C_VEL
LIN {X 0,Y 269.919,Z 449.19,A -85,B 0,C 180,E1 -18313.522,E2 -18313.522} C_VEL
LIN {X 0,Y 265.062,Z 436.896,A -85,B 0,C 180,E1 -18315.095,E2 -18315.095} C_VEL
LIN {X 0,Y 263.676,Z 434.074,A -85,B 0,C 180,E1 -18315.468,E2 -18315.468} C_VEL
LIN {X 0,Y 263.416,Z 432.807,A -85,B 0,C 180,E1 -18315.619,E2 -18315.619} C_VEL
LIN {X 0,Y 263.699,Z 430.717,A -85,B 0,C 180,E1 -18318.265,E2 -18318.265} C_VEL
LIN {X 0,Y 263.787,Z 428.979,A -85,B 0,C 180,E1 -18320.59,E2 -18320.59} C_VEL
LIN {X 0,Y 263.705,Z 426.549,A -85,B 0,C 180,E1 -18324.104,E2 -18324.104} C_VEL
LIN {X 0,Y 263.354,Z 424.212,A -85,B 0,C 180,E1 -18327.742,E2 -18327.742} C_VEL
LIN {X 0,Y 263.251,Z 423.137,A -85,B 0,C 180,E1 -18329.52,E2 -18329.52} C_VEL
LIN {X 0,Y 263.198,Z 422.701,A -85,B 0,C 180,E1 -18331.783,E2 -18331.783} C_VEL
LIN {X 0,Y 263.198,Z 422.702,A -85,B 0,C 180,E1 -18335.212,E2 -18335.212} C_VEL
LIN {X 0,Y 263.259,Z 422.692,A -85,B 0,C 180,E1 -18339.693,E2 -18339.693} C_VEL
LIN {X 0,Y 263.341,Z 422.684,A -85,B 0,C 180,E1 -18344.522,E2 -18344.522} C_VEL
LIN {X 0,Y 263.37,Z 422.673,A -85,B 0,C 180,E1 -18349.235,E2 -18349.235} C_VEL
LIN {X 0,Y 263.569,Z 422.656,A -85,B 0,C 180,E1 -18352.339,E2 -18352.339} C_VEL
LIN {X 0,Y 263.748,Z 422.632,A -85,B 0,C 180,E1 -18358.473,E2 -18358.473} C_VEL
LIN {X 0,Y 263.749,Z 422.633,A -85,B 0,C 180,E1 -18361.527,E2 -18361.527} C_VEL
LIN {X 0,Y 263.566,Z 422.646,A -85,B 0,C 180,E1 -18367.662,E2 -18367.662} C_VEL
LIN {X 0,Y 263.371,Z 422.679,A -85,B 0,C 180,E1 -18370.766,E2 -18370.766} C_VEL
LIN {X 0,Y 263.348,Z 422.682,A -85,B 0,C 180,E1 -18375.478,E2 -18375.478} C_VEL
LIN {X 0,Y 263.261,Z 422.696,A -85,B 0,C 180,E1 -18380.307,E2 -18380.307} C_VEL
LIN {X 0,Y 263.181,Z 422.704,A -85,B 0,C 180,E1 -18383.875,E2 -18383.875} C_VEL
LIN {X 0,Y 262.52,Z 422.788,A -85,B 0,C 180,E1 -18385.153,E2 -18385.153} C_VEL
LIN {X 0,Y 259.643,Z 423.145,A -85,B 0,C 180,E1 -18387.235,E2 -18387.235} C_VEL
LIN {X 0,Y 257.195,Z 423.45,A -85,B 0,C 180,E1 -18388.929,E2 -18388.929} C_VEL
LIN {X 0,Y 256.15,Z 423.579,A -85,B 0,C 180,E1 -18390.243,E2 -18390.243} C_VEL
LIN {X 0,Y 256.068,Z 423.585,A -85,B 0,C 180,E1 -18390.688,E2 -18390.688} C_VEL
LIN {X 0,Y 256.066,Z 423.59,A -85,B 0,C 180,E1 -18393.293,E2 -18393.293} C_VEL
LIN {X 0,Y 256.602,Z 426.143,A -85,B 0,C 180,E1 -18397.414,E2 -18397.414} C_VEL
LIN {X 0,Y 256.987,Z 428.786,A -85,B 0,C 180,E1 -18401.022,E2 -18401.022} C_VEL
LIN {X 0,Y 257.53,Z 432.151,A -85,B 0,C 180,E1 -18405.198,E2 -18405.198} C_VEL
LIN {X 0,Y 257.868,Z 434.016,A -85,B 0,C 180,E1 -18407.381,E2 -18407.381} C_VEL
LIN {X 0,Y 258.243,Z 437.603,A -85,B 0,C 180,E1 -18411.25,E2 -18411.25} C_VEL
LIN {X 0,Y 258.27,Z 439.555,A -85,B 0,C 180,E1 -18413.227,E2 -18413.227} C_VEL
LIN {X 0,Y 258.082,Z 441.517,A -85,B 0,C 180,E1 -18415.12,E2 -18415.12} C_VEL
LIN {X 0,Y 257.525,Z 444.073,A -85,B 0,C 180,E1 -18417.478,E2 -18417.478} C_VEL
LIN {X 0,Y 258.502,Z 447.344,A -85,B 0,C 180,E1 -18417.807,E2 -18417.807} C_VEL
LIN {X 0,Y 262.471,Z 458.685,A -85,B 0,C 180,E1 -18419.174,E2 -18419.174} C_VEL
LIN {X 0,Y 265.676,Z 471.529,A -85,B 0,C 180,E1 -18420.805,E2 -18420.805} C_VEL
LIN {X 0,Y 267.565,Z 482.444,A -85,B 0,C 180,E1 -18422.336,E2 -18422.336} C_VEL
LIN {X 0,Y 268.426,Z 493.445,A -85,B 0,C 180,E1 -18424.029,E2 -18424.029} C_VEL
LIN {X 0,Y 268.325,Z 500.486,A -85,B 0,C 180,E1 -18425.224,E2 -18425.224} C_VEL
LIN {X 0,Y 265.541,Z 510.939,A -85,B 0,C 180,E1 -18427.022,E2 -18427.022} C_VEL
LIN {X 0,Y 263.126,Z 519.438,A -85,B 0,C 180,E1 -18428.864,E2 -18428.864} C_VEL
LIN {X 0,Y 260.731,Z 527.725,A -85,B 0,C 180,E1 -18431.128,E2 -18431.128} C_VEL
LIN {X 0,Y 258.643,Z 534.436,A -85,B 0,C 180,E1 -18433.423,E2 -18433.423} C_VEL
LIN {X 0,Y 256.833,Z 539.825,A -85,B 0,C 180,E1 -18435.743,E2 -18435.743} C_VEL
LIN {X 0,Y 255.637,Z 544.056,A -85,B 0,C 180,E1 -18438.101,E2 -18438.101} C_VEL
LIN {X 0,Y 254.771,Z 547.252,A -85,B 0,C 180,E1 -18440.473,E2 -18440.473} C_VEL
LIN {X 0,Y 254.086,Z 550.061,A -85,B 0,C 180,E1 -18443.648,E2 -18443.648} C_VEL
LIN {X 0,Y 253.975,Z 550.834,A -85,B 0,C 180,E1 -18445.238,E2 -18445.238} C_VEL
LIN {X 0,Y 253.972,Z 551.221,A -85,B 0,C 180,E1 -18446.827,E2 -18446.827} C_VEL
LIN {X 0,Y 254.02,Z 551.225,A -85,B 0,C 180,E1 -18448.414,E2 -18448.414} C_VEL
LIN {X 0,Y 254.057,Z 550.845,A -85,B 0,C 180,E1 -18450,E2 -18450} C_VEL
LIN {X 0,Y 254.052,Z 550.031,A -85,B 0,C 180,E1 -18451.585,E2 -18451.585} C_VEL
LIN {X 0,Y 253.998,Z 548.796,A -85,B 0,C 180,E1 -18453.172,E2 -18453.172} C_VEL
LIN {X 0,Y 254.022,Z 546.743,A -85,B 0,C 180,E1 -18455.118,E2 -18455.118} C_VEL
LIN {X 0,Y 254.309,Z 542.489,A -85,B 0,C 180,E1 -18457.942,E2 -18457.942} C_VEL
LIN {X 0,Y 254.807,Z 537.682,A -85,B 0,C 180,E1 -18460.327,E2 -18460.327} C_VEL
LIN {X 0,Y 255.57,Z 531.588,A -85,B 0,C 180,E1 -18462.708,E2 -18462.708} C_VEL
LIN {X 0,Y 256.877,Z 524.009,A -85,B 0,C 180,E1 -18465.064,E2 -18465.064} C_VEL
LIN {X 0,Y 258.207,Z 516.254,A -85,B 0,C 180,E1 -18467.013,E2 -18467.013} C_VEL
LIN {X 0,Y 259.525,Z 506.747,A -85,B 0,C 180,E1 -18468.963,E2 -18468.963} C_VEL
LIN {X 0,Y 261.116,Z 496.196,A -85,B 0,C 180,E1 -18470.686,E2 -18470.686} C_VEL
LIN {X 0,Y 261.627,Z 492.099,A -85,B 0,C 180,E1 -18471.262,E2 -18471.262} C_VEL
LIN {X 0,Y 260.786,Z 479.557,A -85,B 0,C 180,E1 -18472.892,E2 -18472.892} C_VEL
LIN {X 0,Y 259.392,Z 466.977,A -85,B 0,C 180,E1 -18474.191,E2 -18474.191} C_VEL
LIN {X 0,Y 257.393,Z 454.392,A -85,B 0,C 180,E1 -18475.217,E2 -18475.217} C_VEL
LIN {X 0,Y 255.514,Z 444.886,A -85,B 0,C 180,E1 -18475.848,E2 -18475.848} C_VEL
LIN {X 0,Y 256.518,Z 438.154,A -85,B 0,C 180,E1 -18481.368,E2 -18481.368} C_VEL
LIN {X 0,Y 257.268,Z 433.841,A -85,B 0,C 180,E1 -18485.006,E2 -18485.006} C_VEL
LIN {X 0,Y 257.42,Z 430.826,A -85,B 0,C 180,E1 -18487.65,E2 -18487.65} C_VEL
LIN {X 0,Y 256.826,Z 427.183,A -85,B 0,C 180,E1 -18491.052,E2 -18491.052} C_VEL
LIN {X 0,Y 256.14,Z 423.581,A -85,B 0,C 180,E1 -18494.783,E2 -18494.783} C_VEL
LIN {X 0,Y 256.056,Z 423.593,A -85,B 0,C 180,E1 -18498.796,E2 -18498.796} C_VEL
LIN {X 0,Y 256.127,Z 423.584,A -85,B 0,C 180,E1 -18502.867,E2 -18502.867} C_VEL
LIN {X 0,Y 256.064,Z 423.59,A -85,B 0,C 180,E1 -18506.706,E2 -18506.706} C_VEL
LIN {X 0,Y 256.107,Z 423.58,A -85,B 0,C 180,E1 -18510.399,E2 -18510.399} C_VEL
LIN {X 0,Y 256.184,Z 423.571,A -85,B 0,C 180,E1 -18514.861,E2 -18514.861} C_VEL
LIN {X 0,Y 256.162,Z 423.574,A -85,B 0,C 180,E1 -18519.104,E2 -18519.104} C_VEL
LIN {X 0,Y 256.243,Z 423.547,A -85,B 0,C 180,E1 -18523.724,E2 -18523.724} C_VEL
LIN {X 0,Y 256.285,Z 423.557,A -85,B 0,C 180,E1 -18527.327,E2 -18527.327} C_VEL
LIN {X 0,Y 256.492,Z 423.536,A -85,B 0,C 180,E1 -18530.537,E2 -18530.537} C_VEL
LIN {X 0,Y 256.483,Z 423.529,A -85,B 0,C 180,E1 -18533.707,E2 -18533.707} C_VEL
LIN {X 0,Y 256.709,Z 423.495,A -85,B 0,C 180,E1 -18538.431,E2 -18538.431} C_VEL
LIN {X 0,Y 256.709,Z 423.504,A -85,B 0,C 180,E1 -18541.569,E2 -18541.569} C_VEL
LIN {X 0,Y 256.534,Z 423.526,A -85,B 0,C 180,E1 -18547.873,E2 -18547.873} C_VEL
LIN {X 0,Y 256.304,Z 423.538,A -85,B 0,C 180,E1 -18551.066,E2 -18551.066} C_VEL
LIN {X 0,Y 256.289,Z 423.557,A -85,B 0,C 180,E1 -18555.915,E2 -18555.915} C_VEL
LIN {X 0,Y 256.161,Z 423.572,A -85,B 0,C 180,E1 -18560.895,E2 -18560.895} C_VEL
LIN {X 0,Y 256.183,Z 423.572,A -85,B 0,C 180,E1 -18565.139,E2 -18565.139} C_VEL
LIN {X 0,Y 256.099,Z 423.58,A -85,B 0,C 180,E1 -18569.601,E2 -18569.601} C_VEL
LIN {X 0,Y 256.081,Z 423.585,A -85,B 0,C 180,E1 -18573.291,E2 -18573.291} C_VEL
LIN {X 0,Y 256.137,Z 423.577,A -85,B 0,C 180,E1 -18577.279,E2 -18577.279} C_VEL
LIN {X 0,Y 256.128,Z 423.579,A -85,B 0,C 180,E1 -18581.189,E2 -18581.189} C_VEL
LIN {X 0,Y 256.114,Z 423.584,A -85,B 0,C 180,E1 -18585.517,E2 -18585.517} C_VEL
LIN {X 0,Y 256.13,Z 423.578,A -85,B 0,C 180,E1 -18588.813,E2 -18588.813} C_VEL
LIN {X 0,Y 256.153,Z 423.576,A -85,B 0,C 180,E1 -18592.872,E2 -18592.872} C_VEL
LIN {X 0,Y 256.083,Z 423.585,A -85,B 0,C 180,E1 -18596.711,E2 -18596.711} C_VEL
LIN {X 0,Y 256.137,Z 423.581,A -85,B 0,C 180,E1 -18601.405,E2 -18601.405} C_VEL
LIN {X 0,Y 256.133,Z 423.581,A -85,B 0,C 180,E1 -18605.697,E2 -18605.697} C_VEL
LIN {X 0,Y 256.17,Z 423.591,A -85,B 0,C 180,E1 -18608.557,E2 -18608.557} C_VEL
LIN {X 0,Y 255.666,Z 428.509,A -85,B 0,C 180,E1 -18614.178,E2 -18614.178} C_VEL
LIN {X 0,Y 255.276,Z 432.2,A -85,B 0,C 180,E1 -18618.251,E2 -18618.251} C_VEL
LIN {X 0,Y 258.726,Z 445.496,A -85,B 0,C 180,E1 -18619.262,E2 -18619.262} C_VEL
LIN {X 0,Y 260.778,Z 455.671,A -85,B 0,C 180,E1 -18620.213,E2 -18620.213} C_VEL
LIN {X 0,Y 262.495,Z 467.402,A -85,B 0,C 180,E1 -18621.533,E2 -18621.533} C_VEL
LIN {X 0,Y 263.035,Z 472.196,A -85,B 0,C 180,E1 -18622.153,E2 -18622.153} C_VEL
LIN {X 0,Y 261.675,Z 482.89,A -85,B 0,C 180,E1 -18623.582,E2 -18623.582} C_VEL
LIN {X 0,Y 260.02,Z 493.465,A -85,B 0,C 180,E1 -18625.349,E2 -18625.349} C_VEL
LIN {X 0,Y 258.519,Z 502.626,A -85,B 0,C 180,E1 -18627.273,E2 -18627.273} C_VEL
LIN {X 0,Y 256.999,Z 511.557,A -85,B 0,C 180,E1 -18629.609,E2 -18629.609} C_VEL
LIN {X 0,Y 255.854,Z 518.734,A -85,B 0,C 180,E1 -18631.968,E2 -18631.968} C_VEL
LIN {X 0,Y 255.128,Z 523.58,A -85,B 0,C 180,E1 -18633.949,E2 -18633.949} C_VEL
LIN {X 0,Y 254.582,Z 528.345,A -85,B 0,C 180,E1 -18636.376,E2 -18636.376} C_VEL
LIN {X 0,Y 254.138,Z 531.88,A -85,B 0,C 180,E1 -18638.749,E2 -18638.749} C_VEL
LIN {X 0,Y 253.816,Z 534.46,A -85,B 0,C 180,E1 -18641.176,E2 -18641.176} C_VEL
LIN {X 0,Y 253.771,Z 535.653,A -85,B 0,C 180,E1 -18642.8,E2 -18642.8} C_VEL
LIN {X 0,Y 253.786,Z 536.396,A -85,B 0,C 180,E1 -18644.432,E2 -18644.432} C_VEL
LIN {X 0,Y 253.82,Z 536.746,A -85,B 0,C 180,E1 -18646.075,E2 -18646.075} C_VEL
LIN {X 0,Y 253.962,Z 536.696,A -85,B 0,C 180,E1 -18647.723,E2 -18647.723} C_VEL
LIN {X 0,Y 254.436,Z 535.839,A -85,B 0,C 180,E1 -18650.093,E2 -18650.093} C_VEL
LIN {X 0,Y 255.154,Z 533.906,A -85,B 0,C 180,E1 -18652.682,E2 -18652.682} C_VEL
LIN {X 0,Y 256.155,Z 531.05,A -85,B 0,C 180,E1 -18655.123,E2 -18655.123} C_VEL
LIN {X 0,Y 257.6,Z 526.964,A -85,B 0,C 180,E1 -18657.633,E2 -18657.633} C_VEL
LIN {X 0,Y 259.46,Z 521.263,A -85,B 0,C 180,E1 -18660.251,E2 -18660.251} C_VEL
LIN {X 0,Y 261.984,Z 513.641,A -85,B 0,C 180,E1 -18662.903,E2 -18662.903} C_VEL
LIN {X 0,Y 264.087,Z 506.744,A -85,B 0,C 180,E1 -18664.808,E2 -18664.808} C_VEL
LIN {X 0,Y 266.685,Z 497.665,A -85,B 0,C 180,E1 -18666.836,E2 -18666.836} C_VEL
LIN {X 0,Y 269.465,Z 486.692,A -85,B 0,C 180,E1 -18668.751,E2 -18668.751} C_VEL
LIN {X 0,Y 270.467,Z 481.468,A -85,B 0,C 180,E1 -18669.538,E2 -18669.538} C_VEL
LIN {X 0,Y 269.121,Z 471.513,A -85,B 0,C 180,E1 -18671.225,E2 -18671.225} C_VEL
LIN {X 0,Y 266.505,Z 459.815,A -85,B 0,C 180,E1 -18673.032,E2 -18673.032} C_VEL
LIN {X 0,Y 262.597,Z 447.794,A -85,B 0,C 180,E1 -18674.76,E2 -18674.76} C_VEL
LIN {X 0,Y 257.938,Z 436.79,A -85,B 0,C 180,E1 -18676.282,E2 -18676.282} C_VEL
LIN {X 0,Y 256.677,Z 433.896,A -85,B 0,C 180,E1 -18676.66,E2 -18676.66} C_VEL
LIN {X 0,Y 256.533,Z 433.041,A -85,B 0,C 180,E1 -18676.772,E2 -18676.772} C_VEL
LIN {X 0,Y 256.78,Z 430.61,A -85,B 0,C 180,E1 -18680.026,E2 -18680.026} C_VEL
LIN {X 0,Y 256.749,Z 428.582,A -85,B 0,C 180,E1 -18682.972,E2 -18682.972} C_VEL
LIN {X 0,Y 256.446,Z 426.158,A -85,B 0,C 180,E1 -18686.763,E2 -18686.763} C_VEL
LIN {X 0,Y 256.191,Z 424.032,A -85,B 0,C 180,E1 -18690.41,E2 -18690.41} C_VEL
LIN {X 0,Y 256.139,Z 423.579,A -85,B 0,C 180,E1 -18692.196,E2 -18692.196} C_VEL
LIN {X 0,Y 256.139,Z 423.578,A -85,B 0,C 180,E1 -18695.697,E2 -18695.697} C_VEL
LIN {X 0,Y 256.159,Z 423.579,A -85,B 0,C 180,E1 -18699.105,E2 -18699.105} C_VEL
LIN {X 0,Y 256.277,Z 423.563,A -85,B 0,C 180,E1 -18704.084,E2 -18704.084} C_VEL
LIN {X 0,Y 256.306,Z 423.553,A -85,B 0,C 180,E1 -18708.934,E2 -18708.934} C_VEL
LIN {X 0,Y 256.536,Z 423.53,A -85,B 0,C 180,E1 -18712.127,E2 -18712.127} C_VEL
LIN {X 0,Y 256.711,Z 423.508,A -85,B 0,C 180,E1 -18718.431,E2 -18718.431} C_VEL
LIN {X 0,Y 256.712,Z 423.509,A -85,B 0,C 180,E1 -18721.569,E2 -18721.569} C_VEL
LIN {X 0,Y 256.535,Z 423.523,A -85,B 0,C 180,E1 -18727.873,E2 -18727.873} C_VEL
LIN {X 0,Y 256.307,Z 423.56,A -85,B 0,C 180,E1 -18731.066,E2 -18731.066} C_VEL
LIN {X 0,Y 256.297,Z 423.561,A -85,B 0,C 180,E1 -18735.915,E2 -18735.915} C_VEL
LIN {X 0,Y 256.164,Z 423.579,A -85,B 0,C 180,E1 -18740.896,E2 -18740.896} C_VEL
LIN {X 0,Y 256.187,Z 423.576,A -85,B 0,C 180,E1 -18745.139,E2 -18745.139} C_VEL
LIN {X 0,Y 256.112,Z 423.584,A -85,B 0,C 180,E1 -18749.6,E2 -18749.6} C_VEL
LIN {X 0,Y 256.068,Z 423.585,A -85,B 0,C 180,E1 -18750.688,E2 -18750.688} C_VEL
LIN {X 0,Y 255.432,Z 423.851,A -85,B 0,C 180,E1 -18752.001,E2 -18752.001} C_VEL
LIN {X 0,Y 252.724,Z 425.124,A -85,B 0,C 180,E1 -18754.135,E2 -18754.135} C_VEL
LIN {X 0,Y 250.502,Z 426.508,A -85,B 0,C 180,E1 -18755.863,E2 -18755.863} C_VEL
LIN {X 0,Y 249.665,Z 427.536,A -85,B 0,C 180,E1 -18757.2,E2 -18757.2} C_VEL
LIN {X 0,Y 249.659,Z 427.847,A -85,B 0,C 180,E1 -18757.652,E2 -18757.652} C_VEL
LIN {X 0,Y 250.215,Z 431.275,A -85,B 0,C 180,E1 -18762.385,E2 -18762.385} C_VEL
LIN {X 0,Y 250.806,Z 434.829,A -85,B 0,C 180,E1 -18766.766,E2 -18766.766} C_VEL
LIN {X 0,Y 251.158,Z 437.605,A -85,B 0,C 180,E1 -18769.94,E2 -18769.94} C_VEL
LIN {X 0,Y 251.324,Z 439.558,A -85,B 0,C 180,E1 -18772.034,E2 -18772.034} C_VEL
LIN {X 0,Y 251.16,Z 441.746,A -85,B 0,C 180,E1 -18774.242,E2 -18774.242} C_VEL
LIN {X 0,Y 250.762,Z 443.845,A -85,B 0,C 180,E1 -18776.269,E2 -18776.269} C_VEL
LIN {X 0,Y 251.719,Z 447.124,A -85,B 0,C 180,E1 -18776.619,E2 -18776.619} C_VEL
LIN {X 0,Y 255.147,Z 456.425,A -85,B 0,C 180,E1 -18777.809,E2 -18777.809} C_VEL
LIN {X 0,Y 258.363,Z 468.002,A -85,B 0,C 180,E1 -18779.346,E2 -18779.346} C_VEL
LIN {X 0,Y 260.598,Z 479.219,A -85,B 0,C 180,E1 -18780.959,E2 -18780.959} C_VEL
LIN {X 0,Y 261.756,Z 489.954,A -85,B 0,C 180,E1 -18782.634,E2 -18782.634} C_VEL
LIN {X 0,Y 261.916,Z 500.033,A -85,B 0,C 180,E1 -18784.376,E2 -18784.376} C_VEL
LIN {X 0,Y 261.378,Z 503.344,A -85,B 0,C 180,E1 -18784.945,E2 -18784.945} C_VEL
LIN {X 0,Y 258.503,Z 513.164,A -85,B 0,C 180,E1 -18786.783,E2 -18786.783} C_VEL
LIN {X 0,Y 255.624,Z 522.705,A -85,B 0,C 180,E1 -18789.059,E2 -18789.059} C_VEL
LIN {X 0,Y 253.284,Z 530.326,A -85,B 0,C 180,E1 -18791.392,E2 -18791.392} C_VEL
LIN {X 0,Y 251.155,Z 536.483,A -85,B 0,C 180,E1 -18793.75,E2 -18793.75} C_VEL
LIN {X 0,Y 249.476,Z 541.398,A -85,B 0,C 180,E1 -18796.146,E2 -18796.146} C_VEL
LIN {X 0,Y 248.316,Z 545.214,A -85,B 0,C 180,E1 -18798.573,E2 -18798.573} C_VEL
LIN {X 0,Y 247.311,Z 548.771,A -85,B 0,C 180,E1 -18801.831,E2 -18801.831} C_VEL
LIN {X 0,Y 247.026,Z 549.93,A -85,B 0,C 180,E1 -18803.465,E2 -18803.465} C_VEL
LIN {X 0,Y 246.873,Z 551.029,A -85,B 0,C 180,E1 -18806.736,E2 -18806.736} C_VEL
LIN {X 0,Y 246.928,Z 551.007,A -85,B 0,C 180,E1 -18808.369,E2 -18808.369} C_VEL
LIN {X 0,Y 246.986,Z 550.591,A -85,B 0,C 180,E1 -18810,E2 -18810} C_VEL
LIN {X 0,Y 246.958,Z 549.733,A -85,B 0,C 180,E1 -18811.63,E2 -18811.63} C_VEL
LIN {X 0,Y 246.9,Z 548.47,A -85,B 0,C 180,E1 -18813.263,E2 -18813.263} C_VEL
LIN {X 0,Y 246.952,Z 546.596,A -85,B 0,C 180,E1 -18815.081,E2 -18815.081} C_VEL
LIN {X 0,Y 247.117,Z 543.419,A -85,B 0,C 180,E1 -18817.352,E2 -18817.352} C_VEL
LIN {X 0,Y 247.591,Z 538.945,A -85,B 0,C 180,E1 -18819.806,E2 -18819.806} C_VEL
LIN {X 0,Y 248.293,Z 533.243,A -85,B 0,C 180,E1 -18822.256,E2 -18822.256} C_VEL
LIN {X 0,Y 249.488,Z 526.084,A -85,B 0,C 180,E1 -18824.686,E2 -18824.686} C_VEL
LIN {X 0,Y 250.753,Z 518.786,A -85,B 0,C 180,E1 -18826.695,E2 -18826.695} C_VEL
LIN {X 0,Y 252.197,Z 509.459,A -85,B 0,C 180,E1 -18828.787,E2 -18828.787} C_VEL
LIN {X 0,Y 253.881,Z 498.986,A -85,B 0,C 180,E1 -18830.667,E2 -18830.667} C_VEL
LIN {X 0,Y 254.705,Z 493.822,A -85,B 0,C 180,E1 -18831.444,E2 -18831.444} C_VEL
LIN {X 0,Y 254.135,Z 482.922,A -85,B 0,C 180,E1 -18832.964,E2 -18832.964} C_VEL
LIN {X 0,Y 252.997,Z 471.076,A -85,B 0,C 180,E1 -18834.317,E2 -18834.317} C_VEL
LIN {X 0,Y 251.176,Z 458.306,A -85,B 0,C 180,E1 -18835.488,E2 -18835.488} C_VEL
LIN {X 0,Y 248.728,Z 446.329,A -85,B 0,C 180,E1 -18836.357,E2 -18836.357} C_VEL
LIN {X 0,Y 248.501,Z 444.697,A -85,B 0,C 180,E1 -18836.461,E2 -18836.461} C_VEL
LIN {X 0,Y 249.676,Z 437.77,A -85,B 0,C 180,E1 -18842.331,E2 -18842.331} C_VEL
LIN {X 0,Y 250.357,Z 433.429,A -85,B 0,C 180,E1 -18846.121,E2 -18846.121} C_VEL
LIN {X 0,Y 250.167,Z 430.13,A -85,B 0,C 180,E1 -18849.203,E2 -18849.203} C_VEL
LIN {X 0,Y 249.492,Z 426.375,A -85,B 0,C 180,E1 -18852.911,E2 -18852.911} C_VEL
LIN {X 0,Y 249.07,Z 424.462,A -85,B 0,C 180,E1 -18854.988,E2 -18854.988} C_VEL
LIN {X 0,Y 249.006,Z 424.469,A -85,B 0,C 180,E1 -18859.644,E2 -18859.644} C_VEL
LIN {X 0,Y 249.027,Z 424.465,A -85,B 0,C 180,E1 -18863.654,E2 -18863.654} C_VEL
LIN {X 0,Y 249.034,Z 424.462,A -85,B 0,C 180,E1 -18867.845,E2 -18867.845} C_VEL
LIN {X 0,Y 249.09,Z 424.447,A -85,B 0,C 180,E1 -18871.337,E2 -18871.337} C_VEL
LIN {X 0,Y 249.147,Z 424.448,A -85,B 0,C 180,E1 -18874.968,E2 -18874.968} C_VEL
LIN {X 0,Y 249.105,Z 424.452,A -85,B 0,C 180,E1 -18880.211,E2 -18880.211} C_VEL
LIN {X 0,Y 249.191,Z 424.424,A -85,B 0,C 180,E1 -18883.618,E2 -18883.618} C_VEL
LIN {X 0,Y 249.246,Z 424.439,A -85,B 0,C 180,E1 -18888.616,E2 -18888.616} C_VEL
LIN {X 0,Y 249.479,Z 424.406,A -85,B 0,C 180,E1 -18891.902,E2 -18891.902} C_VEL
LIN {X 0,Y 249.431,Z 424.395,A -85,B 0,C 180,E1 -18896.769,E2 -18896.769} C_VEL
LIN {X 0,Y 249.73,Z 424.369,A -85,B 0,C 180,E1 -18900,E2 -18900} C_VEL
LIN {X 0,Y 249.432,Z 424.412,A -85,B 0,C 180,E1 -18903.23,E2 -18903.23} C_VEL
LIN {X 0,Y 249.475,Z 424.402,A -85,B 0,C 180,E1 -18908.097,E2 -18908.097} C_VEL
LIN {X 0,Y 249.247,Z 424.416,A -85,B 0,C 180,E1 -18911.383,E2 -18911.383} C_VEL
LIN {X 0,Y 249.212,Z 424.441,A -85,B 0,C 180,E1 -18916.503,E2 -18916.503} C_VEL
LIN {X 0,Y 249.082,Z 424.455,A -85,B 0,C 180,E1 -18921.518,E2 -18921.518} C_VEL
LIN {X 0,Y 249.125,Z 424.452,A -85,B 0,C 180,E1 -18925.482,E2 -18925.482} C_VEL
LIN {X 0,Y 249.069,Z 424.453,A -85,B 0,C 180,E1 -18928.99,E2 -18928.99} C_VEL
LIN {X 0,Y 249.032,Z 424.463,A -85,B 0,C 180,E1 -18932.425,E2 -18932.425} C_VEL
LIN {X 0,Y 249.071,Z 424.456,A -85,B 0,C 180,E1 -18936.338,E2 -18936.338} C_VEL
LIN {X 0,Y 249.08,Z 424.456,A -85,B 0,C 180,E1 -18940.463,E2 -18940.463} C_VEL
LIN {X 0,Y 249.09,Z 424.455,A -85,B 0,C 180,E1 -18942.814,E2 -18942.814} C_VEL
LIN {X 0,Y 249.096,Z 424.457,A -85,B 0,C 180,E1 -18947.381,E2 -18947.381} C_VEL
LIN {X 0,Y 249.05,Z 424.463,A -85,B 0,C 180,E1 -18951.625,E2 -18951.625} C_VEL
LIN {X 0,Y 249.059,Z 424.461,A -85,B 0,C 180,E1 -18955.643,E2 -18955.643} C_VEL
LIN {X 0,Y 249.05,Z 424.464,A -85,B 0,C 180,E1 -18959.474,E2 -18959.474} C_VEL
LIN {X 0,Y 249.068,Z 424.461,A -85,B 0,C 180,E1 -18963.163,E2 -18963.163} C_VEL
LIN {X 0,Y 249.058,Z 424.463,A -85,B 0,C 180,E1 -18966.731,E2 -18966.731} C_VEL
LIN {X 0,Y 249.151,Z 424.55,A -85,B 0,C 180,E1 -18968.568,E2 -18968.568} C_VEL
LIN {X 0,Y 248.603,Z 429.162,A -85,B 0,C 180,E1 -18973.982,E2 -18973.982} C_VEL
LIN {X 0,Y 248.257,Z 432.4,A -85,B 0,C 180,E1 -18977.626,E2 -18977.626} C_VEL
LIN {X 0,Y 251.809,Z 445.838,A -85,B 0,C 180,E1 -18978.702,E2 -18978.702} C_VEL
LIN {X 0,Y 253.974,Z 456.464,A -85,B 0,C 180,E1 -18979.739,E2 -18979.739} C_VEL
LIN {X 0,Y 255.692,Z 468.519,A -85,B 0,C 180,E1 -18981.152,E2 -18981.152} C_VEL
LIN {X 0,Y 256.101,Z 474.111,A -85,B 0,C 180,E1 -18981.897,E2 -18981.897} C_VEL
LIN {X 0,Y 254.656,Z 484.482,A -85,B 0,C 180,E1 -18983.361,E2 -18983.361} C_VEL
LIN {X 0,Y 252.956,Z 494.941,A -85,B 0,C 180,E1 -18985.219,E2 -18985.219} C_VEL
LIN {X 0,Y 251.388,Z 503.898,A -85,B 0,C 180,E1 -18987.196,E2 -18987.196} C_VEL
LIN {X 0,Y 249.861,Z 512.641,A -85,B 0,C 180,E1 -18989.597,E2 -18989.597} C_VEL
LIN {X 0,Y 248.742,Z 519.602,A -85,B 0,C 180,E1 -18992.024,E2 -18992.024} C_VEL
LIN {X 0,Y 247.836,Z 525.993,A -85,B 0,C 180,E1 -18994.88,E2 -18994.88} C_VEL
LIN {X 0,Y 247.277,Z 530.198,A -85,B 0,C 180,E1 -18997.348,E2 -18997.348} C_VEL
LIN {X 0,Y 246.853,Z 533.342,A -85,B 0,C 180,E1 -18999.836,E2 -18999.836} C_VEL
LIN {X 0,Y 246.71,Z 534.902,A -85,B 0,C 180,E1 -19001.502,E2 -19001.502} C_VEL
LIN {X 0,Y 246.686,Z 536.544,A -85,B 0,C 180,E1 -19004.386,E2 -19004.386} C_VEL
LIN {X 0,Y 246.761,Z 536.983,A -85,B 0,C 180,E1 -19006.547,E2 -19006.547} C_VEL
LIN {X 0,Y 246.961,Z 536.847,A -85,B 0,C 180,E1 -19008.242,E2 -19008.242} C_VEL
LIN {X 0,Y 247.414,Z 536.055,A -85,B 0,C 180,E1 -19010.382,E2 -19010.382} C_VEL
LIN {X 0,Y 248.283,Z 533.86,A -85,B 0,C 180,E1 -19013.346,E2 -19013.346} C_VEL
LIN {X 0,Y 249.251,Z 531.301,A -85,B 0,C 180,E1 -19015.54,E2 -19015.54} C_VEL
LIN {X 0,Y 250.977,Z 526.662,A -85,B 0,C 180,E1 -19018.427,E2 -19018.427} C_VEL
LIN {X 0,Y 253.251,Z 520.265,A -85,B 0,C 180,E1 -19021.312,E2 -19021.312} C_VEL
LIN {X 0,Y 255.67,Z 513.131,A -85,B 0,C 180,E1 -19023.783,E2 -19023.783} C_VEL
LIN {X 0,Y 258.1,Z 505.63,A -85,B 0,C 180,E1 -19025.834,E2 -19025.834} C_VEL
LIN {X 0,Y 260.724,Z 496.568,A -85,B 0,C 180,E1 -19027.824,E2 -19027.824} C_VEL
LIN {X 0,Y 263.315,Z 486.839,A -85,B 0,C 180,E1 -19029.527,E2 -19029.527} C_VEL
LIN {X 0,Y 264.069,Z 483.294,A -85,B 0,C 180,E1 -19030.076,E2 -19030.076} C_VEL
LIN {X 0,Y 262.724,Z 472.656,A -85,B 0,C 180,E1 -19031.971,E2 -19031.971} C_VEL
LIN {X 0,Y 260.324,Z 461.696,A -85,B 0,C 180,E1 -19033.766,E2 -19033.766} C_VEL
LIN {X 0,Y 256.891,Z 450.894,A -85,B 0,C 180,E1 -19035.44,E2 -19035.44} C_VEL
LIN {X 0,Y 252.907,Z 441.015,A -85,B 0,C 180,E1 -19036.908,E2 -19036.908} C_VEL
LIN {X 0,Y 250.985,Z 436.874,A -85,B 0,C 180,E1 -19037.519,E2 -19037.519} C_VEL
LIN {X 0,Y 249.759,Z 433.953,A -85,B 0,C 180,E1 -19037.916,E2 -19037.916} C_VEL
LIN {X 0,Y 249.636,Z 433.269,A -85,B 0,C 180,E1 -19038.022,E2 -19038.022} C_VEL
LIN {X 0,Y 249.773,Z 430.655,A -85,B 0,C 180,E1 -19041.755,E2 -19041.755} C_VEL
LIN {X 0,Y 249.572,Z 428.128,A -85,B 0,C 180,E1 -19045.723,E2 -19045.723} C_VEL
LIN {X 0,Y 249.277,Z 425.943,A -85,B 0,C 180,E1 -19049.504,E2 -19049.504} C_VEL
LIN {X 0,Y 249.162,Z 424.934,A -85,B 0,C 180,E1 -19051.347,E2 -19051.347} C_VEL
LIN {X 0,Y 249.114,Z 424.454,A -85,B 0,C 180,E1 -19054.525,E2 -19054.525} C_VEL
LIN {X 0,Y 249.09,Z 424.456,A -85,B 0,C 180,E1 -19058.602,E2 -19058.602} C_VEL
LIN {X 0,Y 249.22,Z 424.438,A -85,B 0,C 180,E1 -19063.621,E2 -19063.621} C_VEL
LIN {X 0,Y 249.249,Z 424.433,A -85,B 0,C 180,E1 -19068.617,E2 -19068.617} C_VEL
LIN {X 0,Y 249.478,Z 424.409,A -85,B 0,C 180,E1 -19071.903,E2 -19071.903} C_VEL
LIN {X 0,Y 249.432,Z 424.414,A -85,B 0,C 180,E1 -19076.77,E2 -19076.77} C_VEL
LIN {X 0,Y 249.725,Z 424.379,A -85,B 0,C 180,E1 -19080,E2 -19080} C_VEL
LIN {X 0,Y 249.433,Z 424.415,A -85,B 0,C 180,E1 -19083.231,E2 -19083.231} C_VEL
LIN {X 0,Y 249.477,Z 424.403,A -85,B 0,C 180,E1 -19088.098,E2 -19088.098} C_VEL
LIN {X 0,Y 249.251,Z 424.439,A -85,B 0,C 180,E1 -19091.384,E2 -19091.384} C_VEL
LIN {X 0,Y 249.24,Z 424.442,A -85,B 0,C 180,E1 -19096.379,E2 -19096.379} C_VEL
LIN {X 0,Y 249.085,Z 424.463,A -85,B 0,C 180,E1 -19101.519,E2 -19101.519} C_VEL
LIN {X 0,Y 249.129,Z 424.455,A -85,B 0,C 180,E1 -19105.483,E2 -19105.483} C_VEL
LIN {X 0,Y 249.082,Z 424.461,A -85,B 0,C 180,E1 -19108.994,E2 -19108.994} C_VEL
LIN {X 0,Y 249.029,Z 424.582,A -85,B 0,C 180,E1 -19112.426,E2 -19112.426} C_VEL
LIN {X 0,Y 249.496,Z 426.933,A -85,B 0,C 180,E1 -19116.267,E2 -19116.267} C_VEL
LIN {X 0,Y 249.659,Z 427.847,A -85,B 0,C 180,E1 -19117.652,E2 -19117.652} C_VEL
LIN {X 0,Y 249.202,Z 428.899,A -85,B 0,C 180,E1 -19118.979,E2 -19118.979} C_VEL
LIN {X 0,Y 246.619,Z 431.056,A -85,B 0,C 180,E1 -19121.133,E2 -19121.133} C_VEL
LIN {X 0,Y 244.386,Z 432.865,A -85,B 0,C 180,E1 -19122.883,E2 -19122.883} C_VEL
LIN {X 0,Y 243.505,Z 434.118,A -85,B 0,C 180,E1 -19124.24,E2 -19124.24} C_VEL
LIN {X 0,Y 243.48,Z 434.496,A -85,B 0,C 180,E1 -19124.701,E2 -19124.701} C_VEL
LIN {X 0,Y 244.03,Z 437.62,A -85,B 0,C 180,E1 -19128.518,E2 -19128.518} C_VEL
LIN {X 0,Y 244.214,Z 439.801,A -85,B 0,C 180,E1 -19130.988,E2 -19130.988} C_VEL
LIN {X 0,Y 244.197,Z 442.357,A -85,B 0,C 180,E1 -19133.692,E2 -19133.692} C_VEL
LIN {X 0,Y 243.986,Z 443.821,A -85,B 0,C 180,E1 -19134.981,E2 -19134.981} C_VEL
LIN {X 0,Y 245.023,Z 447.034,A -85,B 0,C 180,E1 -19135.36,E2 -19135.36} C_VEL
LIN {X 0,Y 246.023,Z 449.406,A -85,B 0,C 180,E1 -19135.692,E2 -19135.692} C_VEL
LIN {X 0,Y 249.54,Z 459.411,A -85,B 0,C 180,E1 -19137.086,E2 -19137.086} C_VEL
LIN {X 0,Y 252.645,Z 471.452,A -85,B 0,C 180,E1 -19138.803,E2 -19138.803} C_VEL
LIN {X 0,Y 254.675,Z 483.099,A -85,B 0,C 180,E1 -19140.604,E2 -19140.604} C_VEL
LIN {X 0,Y 255.486,Z 493.576,A -85,B 0,C 180,E1 -19142.373,E2 -19142.373} C_VEL
LIN {X 0,Y 255.273,Z 502.822,A -85,B 0,C 180,E1 -19144.084,E2 -19144.084} C_VEL
LIN {X 0,Y 252.576,Z 511.808,A -85,B 0,C 180,E1 -19145.769,E2 -19145.769} C_VEL
LIN {X 0,Y 249.936,Z 520.068,A -85,B 0,C 180,E1 -19147.691,E2 -19147.691} C_VEL
LIN {X 0,Y 247.331,Z 528.17,A -85,B 0,C 180,E1 -19150.063,E2 -19150.063} C_VEL
LIN {X 0,Y 245.08,Z 534.721,A -85,B 0,C 180,E1 -19152.476,E2 -19152.476} C_VEL
LIN {X 0,Y 243.081,Z 539.968,A -85,B 0,C 180,E1 -19154.917,E2 -19154.917} C_VEL
LIN {X 0,Y 241.717,Z 544.069,A -85,B 0,C 180,E1 -19157.405,E2 -19157.405} C_VEL
LIN {X 0,Y 240.719,Z 547.143,A -85,B 0,C 180,E1 -19159.911,E2 -19159.911} C_VEL
LIN {X 0,Y 240.257,Z 548.688,A -85,B 0,C 180,E1 -19161.59,E2 -19161.59} C_VEL
LIN {X 0,Y 239.802,Z 550.504,A -85,B 0,C 180,E1 -19164.956,E2 -19164.956} C_VEL
LIN {X 0,Y 239.838,Z 550.789,A -85,B 0,C 180,E1 -19168.321,E2 -19168.321} C_VEL
LIN {X 0,Y 239.916,Z 550.324,A -85,B 0,C 180,E1 -19170,E2 -19170} C_VEL
LIN {X 0,Y 239.867,Z 549.435,A -85,B 0,C 180,E1 -19171.679,E2 -19171.679} C_VEL
LIN {X 0,Y 239.842,Z 546.561,A -85,B 0,C 180,E1 -19174.934,E2 -19174.934} C_VEL
LIN {X 0,Y 240.049,Z 543.006,A -85,B 0,C 180,E1 -19177.57,E2 -19177.57} C_VEL
LIN {X 0,Y 240.547,Z 538.468,A -85,B 0,C 180,E1 -19180.096,E2 -19180.096} C_VEL
LIN {X 0,Y 241.295,Z 532.681,A -85,B 0,C 180,E1 -19182.617,E2 -19182.617} C_VEL
LIN {X 0,Y 242.6,Z 525.422,A -85,B 0,C 180,E1 -19185.112,E2 -19185.112} C_VEL
LIN {X 0,Y 243.943,Z 518.03,A -85,B 0,C 180,E1 -19187.175,E2 -19187.175} C_VEL
LIN {X 0,Y 245.299,Z 509.431,A -85,B 0,C 180,E1 -19189.15,E2 -19189.15} C_VEL
LIN {X 0,Y 247.001,Z 499.159,A -85,B 0,C 180,E1 -19191.052,E2 -19191.052} C_VEL
LIN {X 0,Y 247.779,Z 494.028,A -85,B 0,C 180,E1 -19191.855,E2 -19191.855} C_VEL
LIN {X 0,Y 247.241,Z 483.001,A -85,B 0,C 180,E1 -19193.45,E2 -19193.45} C_VEL
LIN {X 0,Y 246.079,Z 470.792,A -85,B 0,C 180,E1 -19194.891,E2 -19194.891} C_VEL
LIN {X 0,Y 244.21,Z 457.8,A -85,B 0,C 180,E1 -19196.122,E2 -19196.122} C_VEL
LIN {X 0,Y 241.537,Z 444.487,A -85,B 0,C 180,E1 -19197.131,E2 -19197.131} C_VEL
LIN {X 0,Y 242.721,Z 437.9,A -85,B 0,C 180,E1 -19202.891,E2 -19202.891} C_VEL
LIN {X 0,Y 243.296,Z 434.421,A -85,B 0,C 180,E1 -19206.018,E2 -19206.018} C_VEL
LIN {X 0,Y 243.21,Z 431.598,A -85,B 0,C 180,E1 -19208.719,E2 -19208.719} C_VEL
LIN {X 0,Y 242.659,Z 428.57,A -85,B 0,C 180,E1 -19211.768,E2 -19211.768} C_VEL
LIN {X 0,Y 242.017,Z 425.34,A -85,B 0,C 180,E1 -19215.39,E2 -19215.39} C_VEL
LIN {X 0,Y 241.954,Z 425.347,A -85,B 0,C 180,E1 -19220.28,E2 -19220.28} C_VEL
LIN {X 0,Y 241.978,Z 425.344,A -85,B 0,C 180,E1 -19224.487,E2 -19224.487} C_VEL
LIN {X 0,Y 241.971,Z 425.344,A -85,B 0,C 180,E1 -19228.479,E2 -19228.479} C_VEL
LIN {X 0,Y 242.003,Z 425.328,A -85,B 0,C 180,E1 -19232.312,E2 -19232.312} C_VEL
LIN {X 0,Y 242.053,Z 425.331,A -85,B 0,C 180,E1 -19236.015,E2 -19236.015} C_VEL
LIN {X 0,Y 242.032,Z 425.332,A -85,B 0,C 180,E1 -19239.607,E2 -19239.607} C_VEL
LIN {X 0,Y 242.15,Z 425.301,A -85,B 0,C 180,E1 -19243.284,E2 -19243.284} C_VEL
LIN {X 0,Y 242.179,Z 425.316,A -85,B 0,C 180,E1 -19248.279,E2 -19248.279} C_VEL
LIN {X 0,Y 242.43,Z 425.284,A -85,B 0,C 180,E1 -19251.665,E2 -19251.665} C_VEL
LIN {X 0,Y 242.256,Z 425.293,A -85,B 0,C 180,E1 -19255.007,E2 -19255.007} C_VEL
LIN {X 0,Y 242.631,Z 425.245,A -85,B 0,C 180,E1 -19258.34,E2 -19258.34} C_VEL
LIN {X 0,Y 242.632,Z 425.257,A -85,B 0,C 180,E1 -19261.66,E2 -19261.66} C_VEL
LIN {X 0,Y 242.423,Z 425.282,A -85,B 0,C 180,E1 -19266.73,E2 -19266.73} C_VEL
LIN {X 0,Y 242.309,Z 425.284,A -85,B 0,C 180,E1 -19270.022,E2 -19270.022} C_VEL
LIN {X 0,Y 242.158,Z 425.314,A -85,B 0,C 180,E1 -19275.141,E2 -19275.141} C_VEL
LIN {X 0,Y 242.067,Z 425.331,A -85,B 0,C 180,E1 -19278.624,E2 -19278.624} C_VEL
LIN {X 0,Y 242.008,Z 425.336,A -85,B 0,C 180,E1 -19282.18,E2 -19282.18} C_VEL
LIN {X 0,Y 242.062,Z 425.335,A -85,B 0,C 180,E1 -19285.838,E2 -19285.838} C_VEL
LIN {X 0,Y 242.003,Z 425.335,A -85,B 0,C 180,E1 -19289.584,E2 -19289.584} C_VEL
LIN {X 0,Y 241.987,Z 425.342,A -85,B 0,C 180,E1 -19293.491,E2 -19293.491} C_VEL
LIN {X 0,Y 242.009,Z 425.338,A -85,B 0,C 180,E1 -19297.578,E2 -19297.578} C_VEL
LIN {X 0,Y 242.033,Z 425.336,A -85,B 0,C 180,E1 -19301.902,E2 -19301.902} C_VEL
LIN {X 0,Y 242.022,Z 425.335,A -85,B 0,C 180,E1 -19306.549,E2 -19306.549} C_VEL
LIN {X 0,Y 242.008,Z 425.338,A -85,B 0,C 180,E1 -19310.292,E2 -19310.292} C_VEL
LIN {X 0,Y 242.034,Z 425.334,A -85,B 0,C 180,E1 -19314.498,E2 -19314.498} C_VEL
LIN {X 0,Y 241.974,Z 425.342,A -85,B 0,C 180,E1 -19318.481,E2 -19318.481} C_VEL
LIN {X 0,Y 242.005,Z 425.338,A -85,B 0,C 180,E1 -19322.313,E2 -19322.313} C_VEL
LIN {X 0,Y 242.037,Z 425.336,A -85,B 0,C 180,E1 -19326.015,E2 -19326.015} C_VEL
LIN {X 0,Y 242.112,Z 425.432,A -85,B 0,C 180,E1 -19328.48,E2 -19328.48} C_VEL
LIN {X 0,Y 241.549,Z 429.81,A -85,B 0,C 180,E1 -19333.77,E2 -19333.77} C_VEL
LIN {X 0,Y 241.212,Z 432.562,A -85,B 0,C 180,E1 -19336.964,E2 -19336.964} C_VEL
LIN {X 0,Y 244.991,Z 446.668,A -85,B 0,C 180,E1 -19338.154,E2 -19338.154} C_VEL
LIN {X 0,Y 247.33,Z 458.266,A -85,B 0,C 180,E1 -19339.352,E2 -19339.352} C_VEL
LIN {X 0,Y 248.931,Z 469.961,A -85,B 0,C 180,E1 -19340.798,E2 -19340.798} C_VEL
LIN {X 0,Y 249.286,Z 474.609,A -85,B 0,C 180,E1 -19341.45,E2 -19341.45} C_VEL
LIN {X 0,Y 247.902,Z 484.332,A -85,B 0,C 180,E1 -19342.86,E2 -19342.86} C_VEL
LIN {X 0,Y 246.198,Z 494.444,A -85,B 0,C 180,E1 -19344.677,E2 -19344.677} C_VEL
LIN {X 0,Y 244.582,Z 503.515,A -85,B 0,C 180,E1 -19346.706,E2 -19346.706} C_VEL
LIN {X 0,Y 242.97,Z 512.368,A -85,B 0,C 180,E1 -19349.172,E2 -19349.172} C_VEL
LIN {X 0,Y 241.765,Z 519.447,A -85,B 0,C 180,E1 -19351.666,E2 -19351.666} C_VEL
LIN {X 0,Y 240.879,Z 525.099,A -85,B 0,C 180,E1 -19354.183,E2 -19354.183} C_VEL
LIN {X 0,Y 240.292,Z 529.55,A -85,B 0,C 180,E1 -19356.719,E2 -19356.719} C_VEL
LIN {X 0,Y 239.99,Z 531.91,A -85,B 0,C 180,E1 -19358.42,E2 -19358.42} C_VEL
LIN {X 0,Y 239.739,Z 533.842,A -85,B 0,C 180,E1 -19360.131,E2 -19360.131} C_VEL
LIN {X 0,Y 239.587,Z 535.302,A -85,B 0,C 180,E1 -19361.849,E2 -19361.849} C_VEL
LIN {X 0,Y 239.584,Z 536.747,A -85,B 0,C 180,E1 -19364.529,E2 -19364.529} C_VEL
LIN {X 0,Y 239.705,Z 537.205,A -85,B 0,C 180,E1 -19367.049,E2 -19367.049} C_VEL
LIN {X 0,Y 239.957,Z 536.977,A -85,B 0,C 180,E1 -19368.794,E2 -19368.794} C_VEL
LIN {X 0,Y 240.378,Z 536.281,A -85,B 0,C 180,E1 -19370.677,E2 -19370.677} C_VEL
LIN {X 0,Y 240.822,Z 535.3,A -85,B 0,C 180,E1 -19372.295,E2 -19372.295} C_VEL
LIN {X 0,Y 241.446,Z 533.777,A -85,B 0,C 180,E1 -19374.048,E2 -19374.048} C_VEL
LIN {X 0,Y 242.687,Z 530.758,A -85,B 0,C 180,E1 -19376.578,E2 -19376.578} C_VEL
LIN {X 0,Y 244.426,Z 526.332,A -85,B 0,C 180,E1 -19379.262,E2 -19379.262} C_VEL
LIN {X 0,Y 246.534,Z 520.749,A -85,B 0,C 180,E1 -19381.828,E2 -19381.828} C_VEL
LIN {X 0,Y 249.049,Z 513.685,A -85,B 0,C 180,E1 -19384.359,E2 -19384.359} C_VEL
LIN {X 0,Y 251.549,Z 506.41,A -85,B 0,C 180,E1 -19386.42,E2 -19386.42} C_VEL
LIN {X 0,Y 254.301,Z 497.506,A -85,B 0,C 180,E1 -19388.449,E2 -19388.449} C_VEL
LIN {X 0,Y 257.084,Z 487.509,A -85,B 0,C 180,E1 -19390.256,E2 -19390.256} C_VEL
LIN {X 0,Y 257.558,Z 485.745,A -85,B 0,C 180,E1 -19390.538,E2 -19390.538} C_VEL
LIN {X 0,Y 257.11,Z 479.339,A -85,B 0,C 180,E1 -19391.757,E2 -19391.757} C_VEL
LIN {X 0,Y 255.684,Z 470.197,A -85,B 0,C 180,E1 -19393.406,E2 -19393.406} C_VEL
LIN {X 0,Y 253.052,Z 459.678,A -85,B 0,C 180,E1 -19395.192,E2 -19395.192} C_VEL
LIN {X 0,Y 248.997,Z 448.021,A -85,B 0,C 180,E1 -19397.084,E2 -19397.084} C_VEL
LIN {X 0,Y 244.431,Z 437.56,A -85,B 0,C 180,E1 -19398.741,E2 -19398.741} C_VEL
LIN {X 0,Y 242.945,Z 434.524,A -85,B 0,C 180,E1 -19399.223,E2 -19399.223} C_VEL
LIN {X 0,Y 242.752,Z 433.519,A -85,B 0,C 180,E1 -19399.365,E2 -19399.365} C_VEL
LIN {X 0,Y 242.744,Z 431.423,A -85,B 0,C 180,E1 -19402.555,E2 -19402.555} C_VEL
LIN {X 0,Y 242.686,Z 430.135,A -85,B 0,C 180,E1 -19404.607,E2 -19404.607} C_VEL
LIN {X 0,Y 242.365,Z 427.871,A -85,B 0,C 180,E1 -19408.537,E2 -19408.537} C_VEL
LIN {X 0,Y 242.086,Z 425.878,A -85,B 0,C 180,E1 -19412.323,E2 -19412.323} C_VEL
LIN {X 0,Y 242.065,Z 425.331,A -85,B 0,C 180,E1 -19414.183,E2 -19414.183} C_VEL
LIN {X 0,Y 242.023,Z 425.335,A -85,B 0,C 180,E1 -19418.313,E2 -19418.313} C_VEL
LIN {X 0,Y 242.161,Z 425.316,A -85,B 0,C 180,E1 -19423.278,E2 -19423.278} C_VEL
LIN {X 0,Y 242.183,Z 425.315,A -85,B 0,C 180,E1 -19428.28,E2 -19428.28} C_VEL
LIN {X 0,Y 242.424,Z 425.287,A -85,B 0,C 180,E1 -19431.666,E2 -19431.666} C_VEL
LIN {X 0,Y 242.256,Z 425.308,A -85,B 0,C 180,E1 -19435.007,E2 -19435.007} C_VEL
LIN {X 0,Y 242.633,Z 425.262,A -85,B 0,C 180,E1 -19438.34,E2 -19438.34} C_VEL
LIN {X 0,Y 242.634,Z 425.263,A -85,B 0,C 180,E1 -19441.66,E2 -19441.66} C_VEL
LIN {X 0,Y 242.429,Z 425.282,A -85,B 0,C 180,E1 -19446.659,E2 -19446.659} C_VEL
LIN {X 0,Y 242.312,Z 425.301,A -85,B 0,C 180,E1 -19450.022,E2 -19450.022} C_VEL
LIN {X 0,Y 242.165,Z 425.322,A -85,B 0,C 180,E1 -19455.141,E2 -19455.141} C_VEL
LIN {X 0,Y 242.071,Z 425.335,A -85,B 0,C 180,E1 -19458.625,E2 -19458.625} C_VEL
LIN {X 0,Y 242.011,Z 425.342,A -85,B 0,C 180,E1 -19462.18,E2 -19462.18} C_VEL
LIN {X 0,Y 242.065,Z 425.335,A -85,B 0,C 180,E1 -19465.839,E2 -19465.839} C_VEL
LIN {X 0,Y 242.029,Z 425.338,A -85,B 0,C 180,E1 -19469.581,E2 -19469.581} C_VEL
LIN {X 0,Y 242.031,Z 425.675,A -85,B 0,C 180,E1 -19471.512,E2 -19471.512} C_VEL
LIN {X 0,Y 242.507,Z 428.159,A -85,B 0,C 180,E1 -19475.763,E2 -19475.763} C_VEL
LIN {X 0,Y 242.897,Z 430.663,A -85,B 0,C 180,E1 -19479.535,E2 -19479.535} C_VEL
LIN {X 0,Y 243.391,Z 433.779,A -85,B 0,C 180,E1 -19483.791,E2 -19483.791} C_VEL
LIN {X 0,Y 243.48,Z 434.496,A -85,B 0,C 180,E1 -19484.701,E2 -19484.701} C_VEL
LIN {X 0,Y 243.01,Z 435.707,A -85,B 0,C 180,E1 -19486.057,E2 -19486.057} C_VEL
LIN {X 0,Y 240.488,Z 438.046,A -85,B 0,C 180,E1 -19488.261,E2 -19488.261} C_VEL
LIN {X 0,Y 237.498,Z 440.945,A -85,B 0,C 180,E1 -19490.968,E2 -19490.968} C_VEL
LIN {X 0,Y 237.192,Z 441.841,A -85,B 0,C 180,E1 -19491.906,E2 -19491.906} C_VEL
LIN {X 0,Y 237.224,Z 443.511,A -85,B 0,C 180,E1 -19493.572,E2 -19493.572} C_VEL
LIN {X 0,Y 238.18,Z 446.593,A -85,B 0,C 180,E1 -19493.951,E2 -19493.951} C_VEL
LIN {X 0,Y 239.338,Z 449.168,A -85,B 0,C 180,E1 -19494.351,E2 -19494.351} C_VEL
LIN {X 0,Y 243.199,Z 459.778,A -85,B 0,C 180,E1 -19495.949,E2 -19495.949} C_VEL
LIN {X 0,Y 246.116,Z 471.151,A -85,B 0,C 180,E1 -19497.667,E2 -19497.667} C_VEL
LIN {X 0,Y 248.198,Z 482.906,A -85,B 0,C 180,E1 -19499.572,E2 -19499.572} C_VEL
LIN {X 0,Y 249.05,Z 492.913,A -85,B 0,C 180,E1 -19501.333,E2 -19501.333} C_VEL
LIN {X 0,Y 248.955,Z 502.347,A -85,B 0,C 180,E1 -19503.149,E2 -19503.149} C_VEL
LIN {X 0,Y 247.99,Z 506.554,A -85,B 0,C 180,E1 -19503.943,E2 -19503.943} C_VEL
LIN {X 0,Y 244.979,Z 515.696,A -85,B 0,C 180,E1 -19505.87,E2 -19505.87} C_VEL
LIN {X 0,Y 242.077,Z 524.298,A -85,B 0,C 180,E1 -19508.174,E2 -19508.174} C_VEL
LIN {X 0,Y 239.43,Z 531.806,A -85,B 0,C 180,E1 -19510.718,E2 -19510.718} C_VEL
LIN {X 0,Y 237.564,Z 536.703,A -85,B 0,C 180,E1 -19512.792,E2 -19512.792} C_VEL
LIN {X 0,Y 235.687,Z 541.484,A -85,B 0,C 180,E1 -19515.317,E2 -19515.317} C_VEL
LIN {X 0,Y 234.368,Z 545.174,A -85,B 0,C 180,E1 -19517.883,E2 -19517.883} C_VEL
LIN {X 0,Y 233.719,Z 547.094,A -85,B 0,C 180,E1 -19519.606,E2 -19519.606} C_VEL
LIN {X 0,Y 233.223,Z 548.591,A -85,B 0,C 180,E1 -19521.334,E2 -19521.334} C_VEL
LIN {X 0,Y 232.733,Z 550.341,A -85,B 0,C 180,E1 -19524.802,E2 -19524.802} C_VEL
LIN {X 0,Y 232.75,Z 550.564,A -85,B 0,C 180,E1 -19528.269,E2 -19528.269} C_VEL
LIN {X 0,Y 232.847,Z 550.05,A -85,B 0,C 180,E1 -19530,E2 -19530} C_VEL
LIN {X 0,Y 232.777,Z 549.132,A -85,B 0,C 180,E1 -19531.73,E2 -19531.73} C_VEL
LIN {X 0,Y 232.758,Z 546.447,A -85,B 0,C 180,E1 -19534.847,E2 -19534.847} C_VEL
LIN {X 0,Y 233.003,Z 542.578,A -85,B 0,C 180,E1 -19537.8,E2 -19537.8} C_VEL
LIN {X 0,Y 233.527,Z 537.967,A -85,B 0,C 180,E1 -19540.402,E2 -19540.402} C_VEL
LIN {X 0,Y 234.522,Z 530.956,A -85,B 0,C 180,E1 -19543.429,E2 -19543.429} C_VEL
LIN {X 0,Y 235.959,Z 523.369,A -85,B 0,C 180,E1 -19545.992,E2 -19545.992} C_VEL
LIN {X 0,Y 237.554,Z 514.461,A -85,B 0,C 180,E1 -19548.386,E2 -19548.386} C_VEL
LIN {X 0,Y 239.337,Z 503.925,A -85,B 0,C 180,E1 -19550.632,E2 -19550.632} C_VEL
LIN {X 0,Y 240.862,Z 494.203,A -85,B 0,C 180,E1 -19552.291,E2 -19552.291} C_VEL
LIN {X 0,Y 240.36,Z 483.306,A -85,B 0,C 180,E1 -19553.934,E2 -19553.934} C_VEL
LIN {X 0,Y 239.201,Z 470.503,A -85,B 0,C 180,E1 -19555.497,E2 -19555.497} C_VEL
LIN {X 0,Y 237.23,Z 457.055,A -85,B 0,C 180,E1 -19556.815,E2 -19556.815} C_VEL
LIN {X 0,Y 234.559,Z 444.271,A -85,B 0,C 180,E1 -19557.825,E2 -19557.825} C_VEL
LIN {X 0,Y 235.766,Z 438.096,A -85,B 0,C 180,E1 -19563.419,E2 -19563.419} C_VEL
LIN {X 0,Y 236.252,Z 434.744,A -85,B 0,C 180,E1 -19566.563,E2 -19566.563} C_VEL
LIN {X 0,Y 236.08,Z 431.991,A -85,B 0,C 180,E1 -19569.284,E2 -19569.284} C_VEL
LIN {X 0,Y 235.347,Z 428.109,A -85,B 0,C 180,E1 -19573.378,E2 -19573.378} C_VEL
LIN {X 0,Y 234.976,Z 426.217,A -85,B 0,C 180,E1 -19575.559,E2 -19575.559} C_VEL
LIN {X 0,Y 234.939,Z 426.224,A -85,B 0,C 180,E1 -19581.055,E2 -19581.055} C_VEL
LIN {X 0,Y 234.924,Z 426.222,A -85,B 0,C 180,E1 -19585.36,E2 -19585.36} C_VEL
LIN {X 0,Y 234.928,Z 426.217,A -85,B 0,C 180,E1 -19589.431,E2 -19589.431} C_VEL
LIN {X 0,Y 234.99,Z 426.204,A -85,B 0,C 180,E1 -19593.793,E2 -19593.793} C_VEL
LIN {X 0,Y 235.007,Z 426.209,A -85,B 0,C 180,E1 -19598.969,E2 -19598.969} C_VEL
LIN {X 0,Y 235.085,Z 426.18,A -85,B 0,C 180,E1 -19603.065,E2 -19603.065} C_VEL
LIN {X 0,Y 235.11,Z 426.195,A -85,B 0,C 180,E1 -19607.921,E2 -19607.921} C_VEL
LIN {X 0,Y 235.386,Z 426.161,A -85,B 0,C 180,E1 -19611.414,E2 -19611.414} C_VEL
LIN {X 0,Y 235.401,Z 426.155,A -85,B 0,C 180,E1 -19613.141,E2 -19613.141} C_VEL
LIN {X 0,Y 235.591,Z 426.12,A -85,B 0,C 180,E1 -19618.29,E2 -19618.29} C_VEL
LIN {X 0,Y 235.591,Z 426.134,A -85,B 0,C 180,E1 -19621.709,E2 -19621.709} C_VEL
LIN {X 0,Y 235.399,Z 426.157,A -85,B 0,C 180,E1 -19626.859,E2 -19626.859} C_VEL
LIN {X 0,Y 235.233,Z 426.161,A -85,B 0,C 180,E1 -19630.326,E2 -19630.326} C_VEL
LIN {X 0,Y 235.106,Z 426.193,A -85,B 0,C 180,E1 -19635.607,E2 -19635.607} C_VEL
LIN {X 0,Y 235.003,Z 426.21,A -85,B 0,C 180,E1 -19639.206,E2 -19639.206} C_VEL
LIN {X 0,Y 234.956,Z 426.213,A -85,B 0,C 180,E1 -19642.883,E2 -19642.883} C_VEL
LIN {X 0,Y 234.963,Z 426.214,A -85,B 0,C 180,E1 -19646.658,E2 -19646.658} C_VEL
LIN {X 0,Y 234.918,Z 426.22,A -85,B 0,C 180,E1 -19650.569,E2 -19650.569} C_VEL
LIN {X 0,Y 234.956,Z 426.213,A -85,B 0,C 180,E1 -19654.633,E2 -19654.633} C_VEL
LIN {X 0,Y 234.963,Z 426.215,A -85,B 0,C 180,E1 -19658.953,E2 -19658.953} C_VEL
LIN {X 0,Y 234.993,Z 426.213,A -85,B 0,C 180,E1 -19663.461,E2 -19663.461} C_VEL
LIN {X 0,Y 234.994,Z 426.21,A -85,B 0,C 180,E1 -19666.54,E2 -19666.54} C_VEL
LIN {X 0,Y 234.952,Z 426.218,A -85,B 0,C 180,E1 -19671.087,E2 -19671.087} C_VEL
LIN {X 0,Y 234.958,Z 426.219,A -85,B 0,C 180,E1 -19675.368,E2 -19675.368} C_VEL
LIN {X 0,Y 234.968,Z 426.215,A -85,B 0,C 180,E1 -19680.158,E2 -19680.158} C_VEL
LIN {X 0,Y 234.993,Z 426.213,A -85,B 0,C 180,E1 -19683.794,E2 -19683.794} C_VEL
LIN {X 0,Y 235.063,Z 426.407,A -85,B 0,C 180,E1 -19688.479,E2 -19688.479} C_VEL
LIN {X 0,Y 234.457,Z 431.158,A -85,B 0,C 180,E1 -19694.349,E2 -19694.349} C_VEL
LIN {X 0,Y 234.229,Z 432.767,A -85,B 0,C 180,E1 -19696.262,E2 -19696.262} C_VEL
LIN {X 0,Y 238.235,Z 447.8,A -85,B 0,C 180,E1 -19697.601,E2 -19697.601} C_VEL
LIN {X 0,Y 240.541,Z 459.02,A -85,B 0,C 180,E1 -19698.825,E2 -19698.825} C_VEL
LIN {X 0,Y 242.09,Z 470.593,A -85,B 0,C 180,E1 -19700.318,E2 -19700.318} C_VEL
LIN {X 0,Y 242.428,Z 475.737,A -85,B 0,C 180,E1 -19701.068,E2 -19701.068} C_VEL
LIN {X 0,Y 240.649,Z 487.314,A -85,B 0,C 180,E1 -19702.868,E2 -19702.868} C_VEL
LIN {X 0,Y 238.769,Z 497.846,A -85,B 0,C 180,E1 -19704.934,E2 -19704.934} C_VEL
LIN {X 0,Y 237.164,Z 506.351,A -85,B 0,C 180,E1 -19707.028,E2 -19707.028} C_VEL
LIN {X 0,Y 235.551,Z 514.646,A -85,B 0,C 180,E1 -19709.573,E2 -19709.573} C_VEL
LIN {X 0,Y 234.449,Z 521.312,A -85,B 0,C 180,E1 -19712.148,E2 -19712.148} C_VEL
LIN {X 0,Y 233.554,Z 527.405,A -85,B 0,C 180,E1 -19715.18,E2 -19715.18} C_VEL
LIN {X 0,Y 233.008,Z 531.373,A -85,B 0,C 180,E1 -19717.801,E2 -19717.801} C_VEL
LIN {X 0,Y 232.595,Z 534.307,A -85,B 0,C 180,E1 -19720.445,E2 -19720.445} C_VEL
LIN {X 0,Y 232.484,Z 535.692,A -85,B 0,C 180,E1 -19722.217,E2 -19722.217} C_VEL
LIN {X 0,Y 232.487,Z 536.949,A -85,B 0,C 180,E1 -19724.682,E2 -19724.682} C_VEL
LIN {X 0,Y 232.671,Z 537.39,A -85,B 0,C 180,E1 -19727.581,E2 -19727.581} C_VEL
LIN {X 0,Y 233.347,Z 536.508,A -85,B 0,C 180,E1 -19730.987,E2 -19730.987} C_VEL
LIN {X 0,Y 233.946,Z 535.29,A -85,B 0,C 180,E1 -19732.988,E2 -19732.988} C_VEL
LIN {X 0,Y 235.49,Z 531.813,A -85,B 0,C 180,E1 -19736.451,E2 -19736.451} C_VEL
LIN {X 0,Y 237.26,Z 527.632,A -85,B 0,C 180,E1 -19739.258,E2 -19739.258} C_VEL
LIN {X 0,Y 239.388,Z 522.368,A -85,B 0,C 180,E1 -19741.9,E2 -19741.9} C_VEL
LIN {X 0,Y 241.973,Z 515.636,A -85,B 0,C 180,E1 -19744.497,E2 -19744.497} C_VEL
LIN {X 0,Y 245.026,Z 507.183,A -85,B 0,C 180,E1 -19747.037,E2 -19747.037} C_VEL
LIN {X 0,Y 247.888,Z 498.454,A -85,B 0,C 180,E1 -19749.11,E2 -19749.11} C_VEL
